(* CoDeSys 2.3.9.59 project: Indo_Tex.pro *)
(* Libraries: standard.lib 5.6.98 12:03:02, TcEtherCAT.lib 8.3.12 17:06:42, TcUtilities.lib 10.1.13 19:12:12, TcBase.lib 14.5.09 12:14:08, FB_Date_Time .lib 20.5.16 16:54:40, TcSystem.lib 27.2.12 14:08:36, TcBaseMath.lib 27.7.04 12:07:56, TcMath.lib 23.9.04 15:15:30, TcMC2.lib 13.9.17 10:18:38, SysLibVisu.lib 7.7.04 17:17:22, SysLibTargetVisu.lib 16.6.08 16:24:26, TcSystemCX.lib 7.9.16 12:51:26, COMlibV2.lib 1.8.08 13:22:48 *)

(* Global variable list: GVL_Alarm *)
VAR_GLOBAL
	RS_Error_1: RS_Error;
	RS_Error_2: RS_Error;
	RS_Error_3: RS_Error;
	RS_Error_4: RS_Error;
	RS_Error_5: RS_Error;
	RS_Error_6: RS_Error;
	RS_Error_7: RS_Error;

	bASealConvEnd1: BOOL;
	AlarmMess2: STRING(80);
	AlarmMess1: STRING(80);
	AlarWrap: STRING(80);
	CountMess: STRING(80);
	AlarmMessg: STRING(80);
	UnitASenSelet: UINT;
	SealingStep: INT;
	AlarmWrpConyMess: STRING(80);
	ConeMissAlarm: STRING(80);

	bAConeFeedCylRsError: BOOL;
	bAFwdCylRsError: BOOL;
	bAWrappingCylRsError: BOOL;
	bAWrappingCylRs1Error: BOOL;
	bAWrappingCylRs2Error: BOOL;
	bAWrappingCylRs3Error: BOOL;
	bAWrapCylRsErrorAuto: BOOL;
	bAError: BOOL;
	bASealTopCylRsError: BOOL;
	bASealBotCylRsError: BOOL;
	bASealTopBotCylRsError: BOOL;
	bASealSepXCylRsError: BOOL;
	bASealSepYCylRsError: BOOL;
	bASupplyPressureError: BOOL;
	HmiSupplyPressureMsg: STRING;
	bAFilmNotloaded: BOOL;
	bAConeMissAtSealConv: BOOL;
	bAEmergencyPressed: BOOL;
	bEmPopUp: BOOL;
	bAConeMissErrorAtWrpConv: BOOL;
	ConeAlignErr: BOOL;
	ConeMissAlarm1: STRING;
	ConeMissAlarm2: STRING;
	bAFlimNotLoaded: BOOL;
	bAPolythinSheetError: BOOL;
	bFilmErrClear: BOOL;
	bASepYAxisRsErrorChkBit: BOOL;
	bASepYAxisRsErrorChkBit1: BOOL;
	bABuzzer: BOOL;
	PressureChkTimer: TON;
	bAStop: BOOL;

	bAErrorChkBit: BOOL;
	bCheckWrappingSen: BOOL;
	bPloySheetSensError: BOOL;
	checkPolySheet2: BOOL;
	bAErrorChkBit2: BOOL;
	bCheckWrappingSen2: BOOL;
	bAErrorChkBit3: BOOL;
	bCheckWrappingSen3: BOOL;
	bWrapConvStopped2Temp: BOOL;
	SealingOk: BOOL;
	CycleComplete: BOOL;
	CycleComplete1: BOOL;
	SGrossWtNokMsg: STRING;

	SGrossWtCylEndSenErrMsg: STRING;
	bGrossWtCylEndSenError: BOOL;
END_VAR

(* Global variable list: GVL_Auto *)
VAR_GLOBAL
	bAutoModeOn: BOOL;
	bAPauseSeq: BOOL;
	bUnitBRowStopperStarted: BOOL;
	bUnitARowStopperStarted: BOOL;
	bAUnitAWeighOk: BOOL;
	bAConeFeedOver: BOOL;
	bAWrappingConvStart3: BOOL;
	bAWrappingConvStart1: BOOL;
	bAWrappingConvStart2: BOOL;
			bA3ConeWrappOver: BOOL;
	bA4thWrappOver: BOOL;
	bA6thConeWrappOver: BOOL;
	bA8thConeWrappOver: BOOL;
	bA6ConeWrappOver23: BOOL;
	AlarmMess: STRING(80);
	bAWrappingCone123OnAuto: BOOL;
	bAFwdPistonComp1: BOOL;
	bAFwdPistonComp2: BOOL;
	bAFwdPistonComp3: BOOL;
	bAConvFirstStart: BOOL;
	UnitACompleteCheckCount: CTU;
	bRetUnitAStart: BOOL;
	bRetUnitBStart: BOOL;
	bAUnitBWeighOk: BOOL;
	(*UnitAConeCompChkCount: CTU;*)
	iSensorOnVal: USINT;
	bFwdPistonStartTemp: BOOL;
	bConeMiss1AtWrapConv: BOOL;
	bConeMiss2tWrapConv: BOOL;
	bConeMiss2AtWrapConv: BOOL;
	ConeMissbit: BOOL;
	CTU_1: CTU;
	bAPauseEnable: BOOL;
	SealComDlyTemp: TIME;
	bAMcStartInAuto: BOOL;
	bPauseExtend: BOOL;
	bAutoModeOff: BOOL;
	iTotalNoOfCones: BOOL;
	iATotalNoOfCones: INT;
	bAMcReady: BOOL;
	bAMcRunninig: BOOL;
	bAFilmLoaded: BOOL;
	bAWrapConStart: BOOL;
	bA3ConeWrappOverTemp: BOOL;
	bABypassOn: BOOL;
	bIntialAckBit: BOOL;
	ConeInComplete: BOOL;
	ConeInCompletetest: BOOL;
	ConeInCompleteTestbitB: BOOL;
	bUnitACounterDIsable: BOOL;
	ConeInCompleteA: BOOL;
	bAOneMinConvStart: BOOL;
	bAWrapwait: BOOL;
END_VAR

(* Global variable list: GVL_Hmi *)
VAR_GLOBAL
	bStopHmi: BOOL;
	bInitializeHmi: BOOL;

	HMIFeedPiston: STRING(80);
	HMIWrapPiston1: STRING(80);
	HMIWrapPiston2: STRING(80);
	HMIWrapPiston3: STRING(80);
	HMIForwdPiston:STRING(80);
	HMISealBotPiston:STRING(80);
	HMISealTopPiston:STRING(80);
	HmiXAxisPiston:STRING(80);
	HmiYAxisPiston:STRING(80);
	bErrorReset: BOOL;
	bPauseHmi: BOOL;
	bResumeHmi: BOOL;
	bResetTemp: BOOL;
	bHmiAck: BOOL;

	b18ConeModelHmi: BOOL;
	b12ConeModelHmi:BOOL;
	b24ConeModelHmi: BOOL;
	b32ConeModelHmi: BOOL;
	sAMcModeStatus: STRING;
	bAUnitBConeCrossed: BOOL;
	bAInializeStarted: BOOL;
	PopUp: BOOL;
	sAlarmStatus: STRING;
	bNegTolDisableHMI: BOOL;
	bNegTolEnableHMI: BOOL;
	bPrssurePopUp: BOOL;
	UnitAConeCountHMI: INT;
	UnitBConeCountHMI: INT;
	b16ConeModelHmi: BOOL;
	WrapConeSenDetMes: STRING;
	bAmberbit2: BOOL;
	Pgm_NoHmi: INT;
	FileCreateTemp: BOOL;
	bACyclePass: BOOL;
	iCartoNoHmi: STRING;
	(*iLotNoHmi: STRING;*)
	var_1: REAL;
	var_5: REAL;
	LogYear: STRING;
	LogMonth: STRING;
	logDay: STRING;
	sTIME: STRING;
	sDATEFinal: STRING;
	DateTimeVar: STRING;
	wTodayToHmi: STRING;
	bInterlockInitial_2: BOOL;
	sMessage: STRING;
	bReadGWieght: BOOL;
	bAReset_all_error: BOOL;








	LotASelected: BOOL;
	LotACartonNo: INT;
	LotBSelected: BOOL;
	LotBCartonNo: INT;
	LotCSelected: BOOL;
	LotDSelected: BOOL;
	LotESelected: BOOL;
	LotFSelected: BOOL;
	LotCCartonNo: INT;
	LotDCartonNo:  INT;
	LotECartonNo:  INT;
	LotFCartonNo: INT;
	LotA: INT;

	LotB: INT;

	LotC: INT;

	LotAHmi: BOOL;
	LotBHmi: BOOL;
	LotCHmi: BOOL;
	CurrentCartonNo:INT;
	LotNoChange: BOOL;
	ParametesSave: BOOL;
END_VAR

VAR_GLOBAL RETAIN
(*VAR_GLOBAL PERSISTENT*)
	b12ConeModelSelected AT %Q*: BOOL;
	b18ConeModelSelected AT %Q*: BOOL;
	b24ConeModelSelected AT %Q*: BOOL;
	b32ConeModelSelected AT %Q*: BOOL;
	rSealCompDlyHmi AT %Q*: REAL;
	iNetTolHmi AT %Q*: REAL;
	iNetWtHmi AT %Q*: REAL;
	iLotNoHmi AT %Q*: STRING;
	iWorkOrderNoHmi AT %Q*:STRING;
	NegToleranceEnabled AT %Q*: BOOL;
	b16ConeModelSelected AT %Q*: BOOL;
	ProgramNoHmi AT %Q*: INT;
	CountCodeHmi AT %Q*: STRING(80);
	CartonNoHmi AT %Q*: INT;
	DefaultNetWeightHmi AT %Q*: REAL;
	DefaultGrossWeightHmi AT %Q*: REAL;
	EmptyConeWt AT %Q*: REAL;
	BlendHmi AT %Q*: STRING(80);
	ShadeHmi AT %Q*: STRING(80);
	ConeTipHmi AT %Q*: STRING(80);
	ConeNettHmi AT %Q*: STRING(80);
	ConeLengthHmi AT %Q*: REAL;
	Cones:INT;
	Dom_ExpHmi AT %Q*: STRING(80);
	PackTypeHmi AT %Q*: STRING(80);
	ItemCodeHmi AT %Q*: STRING(80);
	IssueDesp AT %Q*: STRING(80);
	Location AT %Q*: STRING(80);
	Description AT %Q*: STRING(80);
	Remarks AT %Q*: STRING(80);
	Fyear AT %Q*: STRING(80);
	AvgCount AT %Q*: STRING(80);
	TareWeight AT %Q*: REAL;
	BarCode AT %Q*: STRING(80);
	WorkFlag AT %Q*: STRING(80);
END_VAR

(* Global variable list: GVL_Inputs *)
VAR_GLOBAL


(******************EL1809-1(Main)*********************)

	bIConeFeedingPistonHome AT %IX0.0: BOOL;
	bIConeFeedingPistonEnd AT %IX0.1: BOOL;
	bIConeOrientationTop AT %IX0.2: BOOL;
	bIForwardPistonHome AT %IX0.3: BOOL;
	bIForwardPistonEnd AT %IX0.4: BOOL;
	bIWrappingConeDeductionSen AT %IX0.5: BOOL;
	bISpare1 AT %IX0.6: BOOL;
	bISpare2 AT %IX0.7: BOOL;
	bISpare3 AT %IX1.0: BOOL;
	bIWrappingChannelPiston1_Home AT %IX1.1: BOOL;
	bIWrappingChannelPiston1_End AT %IX1.2: BOOL;
	bIWrappingChannelPiston2_Home AT %IX1.3: BOOL;
	bIWrappingChannelPiston2_End AT %IX1.4: BOOL;
	bIWrappingChannelPiston3_Home AT %IX1.5: BOOL;
	bIWrappingChannelPiston3_End AT %IX1.6: BOOL;
	bIWrappingCone1 AT %IX1.7:BOOL;

(******************EL1809-2(Main)*********************)

	bIWrappingCone2 AT %IX2.0: BOOL;
	bIWrappingCone3 AT %IX2.1: BOOL;
	bIWrappingFilmTensionPlate_1 AT %IX2.2: BOOL;
	bIWrappingFilmTensionPlate_2 AT %IX2.3: BOOL;
	bIWrappingFilmTensionPlate_3 AT %IX2.4: BOOL;
	bISealingTopPistonHome AT %IX2.5: BOOL;
	bISealingTopPistonEnd AT %IX2.6: BOOL;
	bISealingBottomPistonHome AT %IX2.7: BOOL;
	bISealingBottomPistonEnd AT %IX3.0: BOOL;
	bIConeCountSensor AT %IX3.1: BOOL;
	bISealingSeparatorYAxisHome AT %IX3.2: BOOL;
	bISealingSeparatorYAxisEnd AT %IX3.3: BOOL;
	bISealingSeparatorXAxisHome AT %IX3.4: BOOL;
	bISealingSeparatorXAxisEnd AT %IX3.5: BOOL;
	bIManualSealing AT %IX3.6: BOOL;
	bIPressureSwitch  AT %IX3.7: BOOL;

(******************EL1809-3(Main)*********************)

	bISpare4  AT %IX4.0: BOOL;
	bISpare5   AT %IX4.1: BOOL;
	bIUnitA_RowStopperHome   AT %IX4.2: BOOL;
	bIUnitA_RowStopperEnd AT %IX4.3: BOOL;
	bIUnitB_RowStopperHome AT %IX4.4: BOOL;
	bIUnitB_RowStopperEnd AT %IX4.5: BOOL;
	bIUnitA_StartPB AT %IX4.6: BOOL;
	bIUnitB_StartPB AT %IX4.7:BOOL;
	bIUnitAConeDetection4 AT %IX5.0:BOOL;
	bIUnitBConeDetection4 AT %IX5.1:BOOL;
	bIUnitAConeDetection1 AT %IX5.2:BOOL;
	bIUnitAConeDetection2 AT %IX5.3:BOOL;
	bIUnitAConeDetection3 AT %IX5.4:BOOL;
	bIUnitAConeCrossing AT %IX5.5:BOOL;
	bIUnitBConeDetection1 AT %IX5.6:BOOL;
	bIUnitBConeDetection2 AT %IX5.7:BOOL;

(******************EL1809-4(Main)*********************)

	bIUnitBConeDetection3 AT %IX6.0:BOOL;
	bIUnitBConeCrossing AT %IX6.1:BOOL;
	bIAutoManual AT %IX6.2:BOOL;
	bIMCStart AT %IX6.3:BOOL;
	bIMCStop AT %IX6.4:BOOL;
	bIKeySwitch AT %IX6.5:BOOL;
	bIEmergency AT %IX6.6:BOOL;
	bIUnitA_RowStopperMiddle AT %IX6.7:BOOL;

	bIUnitB_RowStopperMiddle AT %IX7.0: BOOL;
	bIGross_Crossing_Input  AT %IX7.1: BOOL;
	bIGross_Weight_Stop AT %IX7.2: BOOL;
	bIGross_Cyl_Home AT %IX7.3: BOOL;
	bIGross_Cyl_End AT %IX7.4: BOOL;
	bISpare12 AT %IX7.5: BOOL;
	bISpare13 AT %IX7.6: BOOL;
	bISpare14 AT %IX7.7: BOOL;
END_VAR

(* Global variable list: GVL_Manual *)
VAR_GLOBAL




		bQMConeFeedingPistonValve :BOOL;
		bQMForwardPistonValve  :BOOL;
		bQMReversePistonValve :BOOL;
		bQMWrappingChannelPistonValve1:BOOL;
		bQMWrappingChannelPistonValve2:BOOL;
		bQMWrappingChannelPistonValve3 :BOOL;
		bQMSealingTopPistonValve :BOOL;
		bQMSealingBottomPistonValve:BOOL;


		bQMFeedingConveyorMotor :BOOL;
		bQMWrappingConveyorMotor :BOOL;
		bQMSealingConveyorMotor :BOOL;
		bQMMatrixConveyorMotor :BOOL;
		bQMFilmRollerMotor1 :BOOL;
		bQMFilmRollerMotor2 :BOOL;
		bQMFilmRollerMotor3 :BOOL;




		bQMRowStopperMotorForward  :BOOL;
		bQMRowStopperMotorReverse:BOOL;
		bQMColumnStopperMotorForward :BOOL;
		bQMColumnStopperMotorReverse:BOOL;
		bQMSealingSeparatorYAxisPistonValve :BOOL;
		bQMSealingSeparatorXAxisPistonValve :BOOL;
		bQMConeTiltingPistonValve :BOOL;
		bQMColumnPushPistonValve:BOOL;

		bQMSeparatorHorizontalPistonValveFwd :BOOL;
		bQMSeparatorVerticalPistonValve :BOOL;
		bQMCartonFeedingPistonValve :BOOL;
		bQMConeEjectionPistonValve :BOOL;
		bQMLengthTightPistonValve :BOOL;
		bQMBreadthTightPistonValve:BOOL;
		bQMEmptyCartonConveyorMotor :BOOL;
		bQMCartonConveyorMotor :BOOL;





		bQMVacuumPistonValve  :BOOL;
		bQMSeparatorHorizontalPistonValveRev  :BOOL;
		bQMSpare1  :BOOL;
		bQMSpare2 :BOOL;


	bQMUnitA_LiftPistonValve:BOOL;
	bQMUnitB_LiftPistonValve: BOOL;
	bQMUnitA_RowStopperMotorForward :BOOL;
	bQMUnitA_RowStopperMotorReverse :BOOL;
	bQMUnitB_RowStopperMotorForward :BOOL;
	bQMUnitB_RowStopperMotorReverse:BOOL;
	bQMUnitC_FullCartonConveyor :BOOL;
	bQMUnitC_LiftPistonValve :BOOL;


	bUA_LiftCylOnHmi: BOOL;
	bUA_LiftCylOffHmi: BOOL;
	bUB_LiftCylOnHmi: BOOL;
	bUB_LiftCylOffHmi: BOOL;
	bUA_RowStopperMotorFwd: BOOL;
	bUA_RowStopperMotorFwdOnHmi: BOOL;
	bUA_RowStopperMotorFwdOffHmi: BOOL;
	bUA_RowStopperMotorRevOnHmi: BOOL;
	bUB_RowStopperMotorFwdOnHmi: BOOL;
	bUB_RowStopperMotorRevOnHmi: BOOL;
	bUC_FullCartonConv: BOOL;
	bUC_FullCartonConvOnHmi: BOOL;
	bUC_FullCartonConvOffHmi: BOOL;
	bUC_LiftCylOnHmi: BOOL;
	bUC_LiftCylOffHmi: BOOL;

	bCFPistonOnHmi: BOOL;
	bCFPistonOffHmi: BOOL;
	bFPValveOnHmi:BOOL;
	bFPValveOffHmi:BOOL;
	bRPValveOnHmi:BOOL;
	bRPValveOffHmi:BOOL;
	bWrappingCPV1OnHmi:BOOL;
	bWrappingCPV1OffHmi:BOOL;
	bWrappingCPV2OnHmi:BOOL;
	bWrappingCPV2OffHmi:BOOL;
	bWrappingCPV3OnHmi:BOOL;
	bWrappingCPV3OffHmi:BOOL;
	bSealingTopPVOnHmi:BOOL;
	bSealingTopPVOffHmi:BOOL;
	bSealingBottomPVOnHmi:BOOL;
	bSealingBottomPVOffHmi:BOOL;
	bFCMotorOnHmi:BOOL;
	bFCMotorOffHmi:BOOL;
	bWCMotorOnHmi:BOOL;
	bWCMotorOffHmi:BOOL;

	bSCMotorOnHmi: BOOL;
	bSCMotorOffHmi: BOOL;
	bMCMotorOnHmi: BOOL;
	bMCMotorOffHmi: BOOL;
	bFRMotor2OnHmi: BOOL;
	bFRMotor2OffHmi: BOOL;
	bFRMotor1OnHmi: BOOL;
	bFRMotor1OffHmi: BOOL;
	bFRMotor3OnHmi: BOOL;
	bFRMotor3OffHmi: BOOL;
	bRSMotorForwardOnHmi: BOOL;
	bRSMotorForwardOffHmi: BOOL;
	bRSMotorRevOnHmi: BOOL;
	bRSMotorRevOffHmi: BOOL;
	bCSMotorFwdOnHmi: BOOL;
	bCSMotorFwdOffHmi: BOOL;
	bCSMotorRevOnHmi: BOOL;
	bCSMotorRevOffHmi: BOOL;
	bSSYAxisPistonValveOnHmi: BOOL;
	bSSYAxisPistonValveOffHmi: BOOL;
	bSSXAxisPistonValveOnHmi: BOOL;
	bSSXAxisPistonValveOffHmi: BOOL;
	bCTPistonValveOnHmi: BOOL;
	bCTPistonValveOffHmi: BOOL;
	bCPushPistonValveOnHmi: BOOL;
	bCPushPistonValveOffHmi: BOOL;
	bSHPistonValveOnHmi: BOOL;
	bSHPistonValveOffHmi: BOOL;
	bSVPistonValveOnHmi: BOOL;
	bSVPistonValveOffHmi: BOOL;
	bCPistonValveOnHmi: BOOL;
	bCPistonValveOffHmi: BOOL;
	bCEPistonValveOnHmi: BOOL;
	bCEPistonValveOffHmi: BOOL;
	bLTPistonValveOnHmi: BOOL;
	bLTPistonValveOffHmi: BOOL;
	bBTightPistonValveOnHmi: BOOL;
	bBTightPistonValveOffHmi: BOOL;
	bECCMotorOnHmi: BOOL;
	bECCMotorOffHmi: BOOL;
	bCCMotorOnHmi: BOOL;
	bCCMotorOffHmi: BOOL;
	bVPValveOnHmi: BOOL;
	bVPValveOffHmi: BOOL;
	bSHPistonValveREVOnHmi: BOOL;
	bSHPistonValveREVOffHmi: BOOL;
	bQMSeparatorHorizontalPistonValveFOR: BOOL;
	bQMColumnPushPistonValveY: BOOL;
	bCPushPistonValveYOnHmi: BOOL;
	bCPushPistonValveYOffHmi: BOOL;
	bMManualSealOn: BOOL;
	bQMLengthPistonValve: BOOL;
	bQMBreathPistonValve: BOOL;
	bQMGrossWtPiston: BOOL;
	bQMRollerConvMotor: BOOL;
	bGWPistonOffHmi1: BOOL;
	bManualModeOn: BOOL;
END_VAR

(* Global variable list: GVL_OutputFlags *)
VAR_GLOBAL



		bQAConeFeedingPistonValve  :BOOL;
		bQAForwardPistonValve  :BOOL;
		bQAWrappingChannelPistonValve1  :BOOL;
		bQAWrappingChannelPistonValve2 :BOOL;
		bQAWrappingChannelPistonValve3:BOOL;
		bQASealingTopPistonValve :BOOL;
		bQASealingBottomPistonValve:BOOL;
		bQASealingSeparatorYAxisPistonValve :BOOL;

		bQASealingSeparatorXAxisPistonValve :BOOL;
		bQAFeedingConveyorMotor :BOOL;
		bQAWrappingConveyorMotor:BOOL;
		bQAFilmRollerMotor1 :BOOL;
		bQAFilmRollerMotor2 :BOOL;
		bQAFilmRollerMotor3 :BOOL;
		bQASealingConveyorMotorFWD :BOOL;







		bQAUnitARowStopperMotorFwd  :BOOL;
		bQAUnitARowStopperMotorRev  :BOOL;
		bQAUnitBRowStopperMotorFwd  :BOOL;
		bQAUnitBRowStopperMotorRev :BOOL;
		bQAUnitAWeightOkLamp :BOOL;
		bQAUnitAWeightNokLamp  :BOOL;
		bQAUnitBWeightOkLamp :BOOL;
		bQAUnitBWeightNokLamp  :BOOL;


		bQABuzzer :BOOL;
		bQASpare1 :BOOL;
		bQASpare2 :BOOL;
		bQASpare3  :BOOL;
		bQASpare4  :BOOL;

	bQAUnitA_RowStopperMotorReverse1: BOOL;
	bQAUnitA_RowStopperMotorForward1: BOOL;
	bQASealingConveyorMotor: BOOL;

	bQASealingConveyor1: BOOL;
	bQAWrappingConveyorMotor1: BOOL;
	bQAWrappingConveyorMotor2: BOOL;
	bQAWrappingConveyorMotor3: BOOL;
	bQAAmber: BOOL;
	bQAGreen: BOOL;
	bQARed: BOOL;
	(*UnitBCompleteCheckCount: CTU;*)
END_VAR

(* Global variable list: GVL_Outputs *)
VAR_GLOBAL

		(*===============EL2809-1(Main) ===========*)


		bQConeFeedingPistonValve AT %QX0.0 :BOOL;
		bQForwardPistonValve AT %QX0.1 :BOOL;
		bQWrappingChannelPistonValve1 AT %QX0.2 :BOOL;
		bQWrappingChannelPistonValve2 AT %QX0.3:BOOL;
		bQWrappingChannelPistonValve3 AT %QX0.4:BOOL;
		bQSealingTopPistonValve AT %QX0.5:BOOL;
		bQSealingBottomPistonValve AT %QX0.6:BOOL;
		bQSealingSeparatorYAxisPistonValve AT %QX0.7:BOOL;

		bQSealingSeparatorXAxisPistonValve  AT %QX1.0:BOOL;
		bQFeedingConveyorMotor AT %QX1.1:BOOL;
		bQWrappingConveyorMotor AT %QX1.2:BOOL;
		bQFilmRollerMotor1 AT %QX1.3:BOOL;
		bQFilmRollerMotor2 AT %QX1.4:BOOL;
		bQFilmRollerMotor3 AT %QX1.5:BOOL;
		bQSealingConveyorMotorFWD AT %QX1.6:BOOL;
		bQUnitARowStopperMotorFwd AT %QX1.7:BOOL;



		(*===============EL2809-2( Main )===========*)



		bQUnitARowStopperMotorRev AT %QX2.0 :BOOL;
		bQUnitBRowStopperMotorFwd AT %QX2.1 :BOOL;
		bQUnitBRowStopperMotorRev AT %QX2.2:BOOL;
		bQUnitAWeightOkLamp  AT %QX2.3:BOOL;
		bQUnitAWeightNokLamp  AT %QX2.4:BOOL;
		bQUnitBWeightOkLamp  AT %QX2.5:BOOL;
		bQUnitBWeightNokLamp  AT %QX2.6:BOOL;
		bQTLGreen AT %QX2.7 :BOOL;

		bQTLAmber AT %QX3.0 :BOOL;
		bQTLRed AT %QX3.1 :BOOL;
		bQBuzzer AT %QX3.2 :BOOL;
		bQGross_Roller_On AT %QX3.3:BOOL;
		bQGross_Cylinder_On AT %QX3.4:BOOL;
		bQSpare3 AT %QX3.5:BOOL;
		bQSpare4  AT %QX3.6:BOOL;
		bQSpare5  AT %QX3.7:BOOL;



		(*===============EL2008-2( Main )===========*)








END_VAR

(* Global variable list: GVL_Reset *)
VAR_GLOBAL
	bQRForwardPistonValve: BOOL;
	bQRWrappingChannelPistonValve2: BOOL;
	bQRWrappingChannelPistonValve3: BOOL;
	bQRSealingTopPistonValve: BOOL;
	bQRSealingSeparatorYAxisPistonValve: BOOL;
	bQRSealingSeparatorXAxisPistonValve: BOOL;
	bQRSealingConveyorMotor: BOOL;
	bQRWrappingChannelPistonValve1: BOOL;
	bQRWrappingConveyorMotor: BOOL;
	bFwdPistonRst: BOOL;
	bARWrappingCone123OnRst: BOOL;

	bAR3ConeWrappOver: BOOL;
	bSaelUnitIntOver: BOOL;
	bWCSStart1: BOOL;
	bAInitializeSeq: BOOL;
	bSealConvIntOver: BOOL;
	sSealConvStatus: STRING;
	sWrapConvStatus: STRING;
	bWrpConvIntOver: BOOL;
END_VAR

(* Global variable list: GVL_Serial *)
VAR_GLOBAL
	rRetUnitBWeight: REAL;
	rRetUnitAWeight: REAL;
	COMin_COMPort AT %I*: EL6inData22B;
	COMOut_COMPort AT %Q*: EL6outData22B;
	TxBuffer1: ComBuffer;
	RxBuffer1: ComBuffer;

	COMin_2_COMport_2 AT %I*: EL6inData22B;
	COMout_2_COMport_2 AT %Q*: EL6outData22B;
	TxBuffer2: ComBuffer;
	RxBuffer2: ComBuffer;

	COMin_3_COMport_3 AT %I*: EL6inData22B;
	COMout_3_COMport_3 AT %Q*: EL6outData22B;
	TxBuffer3: ComBuffer;
	RxBuffer3: ComBuffer;

	COMin_4_COMport_4 AT %I*: EL6inData22B;
	COMout_4_COMport_4 AT %Q*: EL6outData22B;
	TxBuffer4: ComBuffer;
	RxBuffer4: ComBuffer;

	rGrossWeight: REAL;
	bGrossWieghtNokTemp: BOOL;
	bGrossWieghtOk: BOOL;
	bQAGrossWieghtOkIndi: BOOL;
	bGrossWieghtNOk: BOOL;
	GrossWtReedSwBit: BOOL;
	bIGrossWtPistonHome: BOOL;
	bAGrossWtHomeSenRsError: BOOL;
	One_Min_Conv_1: INT;
	rGrossWeighToReport: REAL;
END_VAR

VAR_GLOBAL PERSISTENT
	sGrosswt AT %Q*: REAL;
	sGrossTol AT %Q*: REAL;
END_VAR

(* Global variable list: PARAMETERS *)
VAR_GLOBAL
	SAVE: BOOL;
	TotalCones: DINT;
	iBagCount: DINT;
	LOAD: BOOL;
	sBagNoRep: STRING;
	sDayMonthYearDate: STRING;
	PROCESSCOMPLETE: BOOL;



	PRGNO_LOAD: DINT;
	NegTolEnableHmi AT %Q*: BOOL;
	NegTol1EnableHmi AT %Q*: BOOL;
	NegTol2EnableHmi AT %Q*: BOOL;
	NegTol3EnableHmi AT %Q*: BOOL;
	NegTol4EnableHmi AT %Q*: BOOL;
	NegTol5EnableHmi AT %Q*: BOOL;

	PRGNO_DIS AT %Q*: DINT;
	COUNT_DIS AT %Q*: STRING(80);
	DETAILS_DIS AT %Q*: STRING(80);
	LOTNO_DIS AT %Q*: STRING(80);
	CARTONNO_DIS AT %Q*: DINT;
	WORKORDERNO_DIS:STRING;
	BLEND_DIS:STRING;
	SHADE_DIS:STRING;
	CONETIP_DIS:STRING;
	CONELENGTH_DIS:REAL;
	CONENETWT_DIS:REAL;
	DFLTNETWT_DIS AT %Q*: REAL;
	NETWTTOL_DIS AT %Q*: REAL;
	DFLTGROSSWT_DIS AT %Q*: REAL;
	GROSSWTTOL_DIS AT %Q*: REAL;
	NegTol_DIS AT %Q*: REAL;



	PRGNO AT %Q*: DINT;
	COUNT AT %Q*: STRING(80);
	DETAILS AT %Q*: STRING(80);
	LOTNO AT %Q*: STRING(80);
	CARTONNO AT %Q*: DINT;
	WORKORDERNO:STRING;
	BLEND:STRING;
	SHADE:STRING;
	CONETIP:STRING;
	CONELENGTH:REAL;
	CONENETWT:REAL;
	DFLTNETWT AT %Q*: REAL;
	NETWTTOL AT %Q*: REAL;
	DFLTGROSSWT AT %Q*: REAL;
	GROSSWTTOL AT %Q*: REAL;
	NegTol AT %Q*: REAL;

	PRGNO1 AT %Q*: DINT;
	COUNT1 AT %Q*: STRING(80);
	DETAILS1 AT %Q*: STRING(80);
	LOTNO1 AT %Q*: STRING(80);
	CARTONNO1 AT %Q*: DINT;
	WORKORDERNO1:STRING;
	BLEND1:STRING;
	SHADE1:STRING;
	CONETIP1:STRING;
	CONELENGTH1:REAL;
	CONENETWT1:REAL;
	DFLTNETWT1 AT %Q*: REAL;
	NETWTTOL1 AT %Q*: REAL;
	DFLTGROSSWT1 AT %Q*: REAL;
	GROSSWTTOL1 AT %Q*: REAL;
	NegTol1 AT %Q*: REAL;

	PRGNO2 AT %Q*: DINT;
	COUNT2 AT %Q*: STRING(80);
	DETAILS2 AT %Q*: STRING(80);
	LOTNO2 AT %Q*: STRING(80);
	CARTONNO2 AT %Q*: DINT;
	WORKORDERNO2:STRING;
	BLEND2:STRING;
	SHADE2:STRING;
	CONETIP2:STRING;
	CONELENGTH2:REAL;
	CONENETWT2:REAL;
	DFLTNETWT2 AT %Q*: REAL;
	NETWTTOL2 AT %Q*: REAL;
	DFLTGROSSWT2 AT %Q*: REAL;
	GROSSWTTOL2 AT %Q*: REAL;
	NegTol2 AT %Q*: REAL;

	PRGNO3 AT %Q*: DINT;
	COUNT3 AT %Q*: STRING(80);
	DETAILS3 AT %Q*: STRING(80);
	LOTNO3 AT %Q*: STRING(80);
	CARTONNO3 AT %Q*: DINT;
	WORKORDERNO3:STRING;
	BLEND3:STRING;
	SHADE3:STRING;
	CONETIP3:STRING;
	CONELENGTH3:REAL;
	CONENETWT3:REAL;
	DFLTNETWT3 AT %Q*: REAL;
	NETWTTOL3 AT %Q*: REAL;
	DFLTGROSSWT3 AT %Q*: REAL;
	GROSSWTTOL3 AT %Q*: REAL;
	NegTol3 AT %Q*: REAL;

	PRGNO4 AT %Q*: DINT;
	COUNT4 AT %Q*: STRING(80);
	DETAILS4 AT %Q*: STRING(80);
	LOTNO4 AT %Q*: STRING(80);
	CARTONNO4 AT %Q*: DINT;
	WORKORDERNO4:STRING;
	BLEND4:STRING;
	SHADE4:STRING;
	CONETIP4:STRING;
	CONELENGTH4:REAL;
	CONENETWT4:REAL;
	DFLTNETWT4 AT %Q*: REAL;
	NETWTTOL4 AT %Q*: REAL;
	DFLTGROSSWT4 AT %Q*: REAL;
	GROSSWTTOL4 AT %Q*: REAL;
	NegTol4 AT %Q*: REAL;


	PRGNO5 AT %Q*: DINT;
	COUNT5 AT %Q*: STRING(80);
	DETAILS5 AT %Q*: STRING(80);
	LOTNO5 AT %Q*: STRING(80);
	CARTONNO5 AT %Q*: DINT;
	WORKORDERNO5:STRING;
	BLEND5:STRING;
	SHADE5:STRING;
	CONETIP5:STRING;
	CONELENGTH5:REAL;
	CONENETWT5:REAL;
	DFLTNETWT5 AT %Q*: REAL;
	NETWTTOL5 AT %Q*: REAL;
	DFLTGROSSWT5 AT %Q*: REAL;
	GROSSWTTOL5 AT %Q*: REAL;
	NegTol5 AT %Q*: REAL;


	PRGNO6:DINT;
	COUNT6:STRING;
	DETAILS6:STRING;
	LOTNO6:STRING;
	CARTONNO6:DINT;
	WORKORDERNO6:STRING;
	BLEND6:STRING;
	SHADE6:STRING;
	CONETIP6:STRING;
	CONELENGTH6:REAL;
	CONENETWT6:REAL;
	DFLTNETWT6:REAL;
	NETWTTOL6:REAL;
	DFLTGROSSWT6:REAL;
	GROSSWTTOL6:REAL;


	PRGNO7:DINT;
	COUNT7:STRING;
	DETAILS7:STRING;
	LOTNO7:STRING;
	CARTONNO7:DINT;
	WORKORDERNO7:STRING;
	BLEND7:STRING;
	SHADE7:STRING;
	CONETIP7:STRING;
	CONELENGTH7:REAL;
	CONENETWT7:REAL;
	DFLTNETWT7:REAL;
	NETWTTOL7:REAL;
	DFLTGROSSWT7:REAL;
	GROSSWTTOL7:REAL;


	PRGNO8:DINT;
	COUNT8:STRING;
	DETAILS8:STRING;
	LOTNO8:STRING;
	CARTONNO8:DINT;
	WORKORDERNO8:STRING;
	BLEND8:STRING;
	SHADE8:STRING;
	CONETIP8:STRING;
	CONELENGTH8:REAL;
	CONENETWT8:REAL;
	DFLTNETWT8:REAL;
	NETWTTOL8:REAL;
	DFLTGROSSWT8:REAL;
	GROSSWTTOL8:REAL;


	PRGNO9:DINT;
	COUNT9:STRING;
	DETAILS9:STRING;
	LOTNO9:STRING;
	CARTONNO9:DINT;
	WORKORDERNO9:STRING;
	BLEND9:STRING;
	SHADE9:STRING;
	CONETIP9:STRING;
	CONELENGTH9:REAL;
	CONENETWT9:REAL;
	DFLTNETWT9:REAL;
	NETWTTOL9:REAL;
	DFLTGROSSWT9:REAL;
	GROSSWTTOL9:REAL;


	PRGNO10:DINT;
	COUNT10:STRING;
	DETAILS10:STRING;
	LOTNO10:STRING;
	CARTONNO10:DINT;
	WORKORDERNO10:STRING;
	BLEND10:STRING;
	SHADE10:STRING;
	CONETIP10:STRING;
	CONELENGTH10:REAL;
	CONENETWT10:REAL;
	DFLTNETWT10:REAL;
	NETWTTOL10:REAL;
	DFLTGROSSWT10:REAL;
	GROSSWTTOL10:REAL;

	PRG1RUNNING AT %Q*: BOOL;
	PRG2RUNNING AT %Q*: BOOL;
	PRG3RUNNING AT %Q*: BOOL;
	PRG4RUNNING AT %Q*: BOOL;
	PRG5RUNNING AT %Q*: BOOL;
	PRG6RUNNING: BOOL;
	PRG7RUNNING: BOOL;
	PRG8RUNNING: BOOL;
	PRG9RUNNING: BOOL;
	PRG10RUNNING: BOOL;
	PRINTENABLE: BOOL;
	PRINTENABLED: BOOL;

	DfltWtPrint: BOOL;
	DfltGrossWtPrint_En: BOOL;
	GrossWtPrintDflt: BOOL;
	NetwtPrint: STRING;
	GrosswtPrint: STRING;

	ReportPath: STRING;
	sDayF1: STRING;
	sMonthF1: STRING;
	sDayMonth1: STRING;

	ReportPath_Final_2: STRING;
	FB_DateTime_2: FB_DateTime;
	sDaateReport: STRING;







	sDayMonthYear1: STRING;

	sDayMonthYear: STRING;
	ReportPath_Final_1: STRING;
	ReportPath_Final: STRING;
END_VAR

(* Global variable list: PRINT *)
VAR_GLOBAL

	ProductionData_Print: STRING(255);
	ProductionDataValues_Print: STRING(255);
	ProductionDataValues_Print_Com:STRING(255);
	PrintOk: BOOL;
	PrintEnableHmi: BOOL;
	PrintValue: INT;
	bANewDay: BOOL;
	ProductionDataValues_IndoPrint: STRING(255);
	ProductionData_IndoPrint: STRING(255);
	ProductionDataError_IndoPrint: STRING(255);

	ProductionData_IndoPrint2:STRING(255);
	ProductionDataError_IndoPrint2:STRING(255);
	ProductionDataValues_IndoPrint_Com:STRING(255);
		ProductionDataValuesError_IndoPrint_Com:STRING(255);
	ProductionData_IndoPrint11 : ProductionData_IndoPrint1;

	SerialNoError: DINT;




	ReportPathError: STRING;
	ReportPath_FinalError: STRING;
	ReportPath_Final_1Error: STRING;
	ReportPath_Final_2Error: STRING;
	stStation1_ProductionData:Production_Data;
	sHourPreFix: STRING;
	sHou: STRING;
	sDayPreFix: STRING;
	sDay: STRING;
	sMonthPreFix: STRING;
	sMonth: STRING;
	sDayF: STRING;
	sMonthF: STRING;
	sDayMonth: STRING;

	SerialNo AT %Q*: DINT;
	BagSerialNo: DINT;
	ReportSave: BOOL;
	wTodayToHmiFinal: STRING;
	Default_NetWeight_Report: STRING;
	Default_GrossWeight_Report: STRING;
	Actual_NetWeight_Report: STRING;
	Actual_GrossWeight_Report: STRING;
	negativetolerance AT %Q*: BOOL;
	DefaultNetWt AT %Q*: REAL;
	NetWtTolRep AT %Q*: REAL;
	DefaultGrossWt AT %Q*: REAL;
	GrossWtTolRep AT %Q*: REAL;


END_VAR

(* Global variable list: TwinCAT_Configuration *)
(* Generated automatically by TwinCAT - (read only) *)
VAR_CONFIG
	.b12ConeModelSelected AT %QX288.0 : BOOL;	(*  ~ {LinkedWith:TIID^Device 3 (NOV/DP-RAM)^Outputs^Model_1} *)
	.b18ConeModelSelected AT %QX288.1 : BOOL;	(*  ~ {LinkedWith:TIID^Device 3 (NOV/DP-RAM)^Outputs^Model_2} *)
	.b24ConeModelSelected AT %QX288.2 : BOOL;	(*  ~ {LinkedWith:TIID^Device 3 (NOV/DP-RAM)^Outputs^Model_3} *)
	.b32ConeModelSelected AT %QX288.3 : BOOL;	(*  ~ {LinkedWith:TIID^Device 3 (NOV/DP-RAM)^Outputs^Model_4} *)
	.rSealCompDlyHmi AT %QB52 : REAL;	(*  ~ {LinkedWith:TIID^Device 3 (NOV/DP-RAM)^Outputs^SealDly} *)
	.iNetTolHmi AT %QB56 : REAL;	(*  ~ {LinkedWith:TIID^Device 3 (NOV/DP-RAM)^Outputs^NetWtTol} *)
	.iNetWtHmi AT %QB60 : REAL;	(*  ~ {LinkedWith:TIID^Device 3 (NOV/DP-RAM)^Outputs^NetWt} *)
	.iLotNoHmi AT %QB64 : STRING(80);	(*  ~ {LinkedWith:TIID^Device 3 (NOV/DP-RAM)^Outputs^Var 339} *)
	.iWorkOrderNoHmi AT %QB148 : STRING(80);	(*  ~ {LinkedWith:TIID^Device 3 (NOV/DP-RAM)^Outputs^WorkOrderHmi} *)
	.NegToleranceEnabled AT %QX288.4 : BOOL;	(*  ~ {LinkedWith:TIID^Device 3 (NOV/DP-RAM)^Outputs^Var 278} *)
	.b16ConeModelSelected AT %QX288.5 : BOOL;
	.ProgramNoHmi AT %QB2276 : INT;	(*  ~ {LinkedWith:TIID^Device 3 (NOV/DP-RAM)^Outputs^PrgNo} *)
	.CountCodeHmi AT %QB2280 : STRING(80);	(*  ~ {LinkedWith:TIID^Device 3 (NOV/DP-RAM)^Outputs^CountCode} *)
	.CartonNoHmi AT %QB2362 : INT;	(*  ~ {LinkedWith:TIID^Device 3 (NOV/DP-RAM)^Outputs^CartonNo} *)
	.DefaultNetWeightHmi AT %QB2364 : REAL;	(*  ~ {LinkedWith:TIID^Device 3 (NOV/DP-RAM)^Outputs^DfltNetWt} *)
	.DefaultGrossWeightHmi AT %QB2368 : REAL;	(*  ~ {LinkedWith:TIID^Device 3 (NOV/DP-RAM)^Outputs^DfltGrossWt} *)
	.EmptyConeWt AT %QB3640 : REAL;	(*  ~ {LinkedWith:TIID^Device 3 (NOV/DP-RAM)^Outputs^EmptyConet} *)
	.BlendHmi AT %QB2372 : STRING(80);	(*  ~ {LinkedWith:TIID^Device 3 (NOV/DP-RAM)^Outputs^Blend} *)
	.ShadeHmi AT %QB2456 : STRING(80);	(*  ~ {LinkedWith:TIID^Device 3 (NOV/DP-RAM)^Outputs^Shade} *)
	.ConeTipHmi AT %QB2540 : STRING(80);	(*  ~ {LinkedWith:TIID^Device 3 (NOV/DP-RAM)^Outputs^ConeTip} *)
	.ConeNettHmi AT %QB2624 : STRING(80);	(*  ~ {LinkedWith:TIID^Device 3 (NOV/DP-RAM)^Outputs^ConeNetWt} *)
	.ConeLengthHmi AT %QB2708 : REAL;	(*  ~ {LinkedWith:TIID^Device 3 (NOV/DP-RAM)^Outputs^ConeLen} *)
	.Dom_ExpHmi AT %QB2712 : STRING(80);	(*  ~ {LinkedWith:TIID^Device 3 (NOV/DP-RAM)^Outputs^Dom} *)
	.PackTypeHmi AT %QB2796 : STRING(80);	(*  ~ {LinkedWith:TIID^Device 3 (NOV/DP-RAM)^Outputs^PackType} *)
	.ItemCodeHmi AT %QB2880 : STRING(80);	(*  ~ {LinkedWith:TIID^Device 3 (NOV/DP-RAM)^Outputs^ItemCode} *)
	.IssueDesp AT %QB2964 : STRING(80);	(*  ~ {LinkedWith:TIID^Device 3 (NOV/DP-RAM)^Outputs^IssueDes} *)
	.Location AT %QB3048 : STRING(80);	(*  ~ {LinkedWith:TIID^Device 3 (NOV/DP-RAM)^Outputs^Location} *)
	.Description AT %QB3132 : STRING(80);	(*  ~ {LinkedWith:TIID^Device 3 (NOV/DP-RAM)^Outputs^Description} *)
	.Remarks AT %QB3216 : STRING(80);	(*  ~ {LinkedWith:TIID^Device 3 (NOV/DP-RAM)^Outputs^Remarks} *)
	.Fyear AT %QB3300 : STRING(80);	(*  ~ {LinkedWith:TIID^Device 3 (NOV/DP-RAM)^Outputs^FYear} *)
	.AvgCount AT %QB3384 : STRING(80);	(*  ~ {LinkedWith:TIID^Device 3 (NOV/DP-RAM)^Outputs^Avg_Count} *)
	.TareWeight AT %QB3468 : REAL;	(*  ~ {LinkedWith:TIID^Device 3 (NOV/DP-RAM)^Outputs^TareWeight} *)
	.BarCode AT %QB3472 : STRING(80);	(*  ~ {LinkedWith:TIID^Device 3 (NOV/DP-RAM)^Outputs^Var 280} *)
	.WorkFlag AT %QB3556 : STRING(80);	(*  ~ {LinkedWith:TIID^Device 3 (NOV/DP-RAM)^Outputs^Var 279} *)
	.COMin_3_COMport_3 AT %IB56 : EL6inData22B;
	.COMout_3_COMport_3 AT %QB232 : EL6outData22B;
	.COMin_4_COMport_4 AT %IB80 : EL6inData22B;
	.COMout_4_COMport_4 AT %QB256 : EL6outData22B;
	.sGrosswt AT %QB280 : REAL;	(*  ~ {LinkedWith:TIID^Device 3 (NOV/DP-RAM)^Outputs^GrossWt} *)
	.sGrossTol AT %QB284 : REAL;	(*  ~ {LinkedWith:TIID^Device 3 (NOV/DP-RAM)^Outputs^GrossWtTol} *)
	.NegTolEnableHmi AT %QX2272.0 : BOOL;
	.NegTol1EnableHmi AT %QX2272.1 : BOOL;
	.NegTol2EnableHmi AT %QX2272.2 : BOOL;
	.NegTol3EnableHmi AT %QX2272.3 : BOOL;
	.NegTol4EnableHmi AT %QX2272.4 : BOOL;
	.NegTol5EnableHmi AT %QX2272.5 : BOOL;
	.PRGNO_DIS AT %QB292 : DINT;
	.COUNT_DIS AT %QB296 : STRING(80);
	.DETAILS_DIS AT %QB380 : STRING(80);
	.LOTNO_DIS AT %QB464 : STRING(80);
	.CARTONNO_DIS AT %QB548 : DINT;
	.DFLTNETWT_DIS AT %QB552 : REAL;
	.NETWTTOL_DIS AT %QB556 : REAL;
	.DFLTGROSSWT_DIS AT %QB560 : REAL;
	.GROSSWTTOL_DIS AT %QB564 : REAL;
	.NegTol_DIS AT %QB568 : REAL;
	.PRGNO AT %QB572 : DINT;
	.COUNT AT %QB576 : STRING(80);
	.DETAILS AT %QB660 : STRING(80);
	.LOTNO AT %QB744 : STRING(80);
	.CARTONNO AT %QB828 : DINT;
	.DFLTNETWT AT %QB832 : REAL;
	.NETWTTOL AT %QB836 : REAL;
	.DFLTGROSSWT AT %QB840 : REAL;
	.GROSSWTTOL AT %QB844 : REAL;
	.NegTol AT %QB848 : REAL;
	.PRGNO1 AT %QB852 : DINT;
	.COUNT1 AT %QB856 : STRING(80);
	.DETAILS1 AT %QB940 : STRING(80);
	.LOTNO1 AT %QB1024 : STRING(80);
	.CARTONNO1 AT %QB1108 : DINT;
	.DFLTNETWT1 AT %QB1112 : REAL;
	.NETWTTOL1 AT %QB1116 : REAL;
	.DFLTGROSSWT1 AT %QB1120 : REAL;
	.GROSSWTTOL1 AT %QB1124 : REAL;
	.NegTol1 AT %QB1128 : REAL;
	.PRGNO2 AT %QB1132 : DINT;
	.COUNT2 AT %QB1136 : STRING(80);
	.DETAILS2 AT %QB1220 : STRING(80);
	.LOTNO2 AT %QB1304 : STRING(80);
	.CARTONNO2 AT %QB1388 : DINT;
	.DFLTNETWT2 AT %QB1392 : REAL;
	.NETWTTOL2 AT %QB1396 : REAL;
	.DFLTGROSSWT2 AT %QB1400 : REAL;
	.GROSSWTTOL2 AT %QB1404 : REAL;
	.NegTol2 AT %QB1408 : REAL;
	.PRGNO3 AT %QB1412 : DINT;
	.COUNT3 AT %QB1416 : STRING(80);
	.DETAILS3 AT %QB1500 : STRING(80);
	.LOTNO3 AT %QB1584 : STRING(80);
	.CARTONNO3 AT %QB1668 : DINT;
	.DFLTNETWT3 AT %QB1672 : REAL;
	.NETWTTOL3 AT %QB1676 : REAL;
	.DFLTGROSSWT3 AT %QB1680 : REAL;
	.GROSSWTTOL3 AT %QB1684 : REAL;
	.NegTol3 AT %QB1688 : REAL;
	.PRGNO4 AT %QB1692 : DINT;
	.COUNT4 AT %QB1696 : STRING(80);
	.DETAILS4 AT %QB1780 : STRING(80);
	.LOTNO4 AT %QB1864 : STRING(80);
	.CARTONNO4 AT %QB1948 : DINT;
	.DFLTNETWT4 AT %QB1952 : REAL;
	.NETWTTOL4 AT %QB1956 : REAL;
	.DFLTGROSSWT4 AT %QB1960 : REAL;
	.GROSSWTTOL4 AT %QB1964 : REAL;
	.NegTol4 AT %QB1968 : REAL;
	.PRGNO5 AT %QB1972 : DINT;
	.COUNT5 AT %QB1976 : STRING(80);
	.DETAILS5 AT %QB2060 : STRING(80);
	.LOTNO5 AT %QB2144 : STRING(80);
	.CARTONNO5 AT %QB2228 : DINT;
	.DFLTNETWT5 AT %QB2232 : REAL;
	.NETWTTOL5 AT %QB2236 : REAL;
	.DFLTGROSSWT5 AT %QB2240 : REAL;
	.GROSSWTTOL5 AT %QB2244 : REAL;
	.NegTol5 AT %QB2248 : REAL;
	.PRG1RUNNING AT %QX2272.6 : BOOL;
	.PRG2RUNNING AT %QX2272.7 : BOOL;
	.PRG3RUNNING AT %QX2273.0 : BOOL;
	.PRG4RUNNING AT %QX2273.1 : BOOL;
	.PRG5RUNNING AT %QX2273.2 : BOOL;
	.SerialNo AT %QB2252 : DINT;
	.negativetolerance AT %QX2273.3 : BOOL;
	.DefaultNetWt AT %QB2256 : REAL;
	.NetWtTolRep AT %QB2260 : REAL;
	.DefaultGrossWt AT %QB2264 : REAL;	(*  ~ {LinkedWith:TIID^Device 3 (NOV/DP-RAM)^Outputs^Var 299} *)
	.GrossWtTolRep AT %QB2268 : REAL;
END_VAR

(* Global variable list: TwinCAT_Configuration_1 *)
(* Generated automatically by TwinCAT - (read only) *)
VAR_CONFIG
	.COMin_COMPort AT %IB8 : EL6inData22B;
	.COMOut_COMPort AT %QB4 : EL6outData22B;
	.COMin_2_COMport_2 AT %IB32 : EL6inData22B;
	.COMout_2_COMport_2 AT %QB28 : EL6outData22B;
END_VAR

(* Data type *)
TYPE Production_Data :
STRUCT

	S_No						:STRING;
	ConeType					:STRING;
	CartonNo					:STRING;
	LotNo						:STRING;
	SDateF						:STRING;
	NetWt						:STRING;
	WorkOrderNo				:STRING;
	DefaultNettWeight				:STRING;
	DefaultGrossWeight			:STRING;
	Blend						:STRING;
	Shade						:STRING;
	ConeTip						:STRING;
	ConeNettWeight				:STRING;
	ConeLength					:STRING;
	Dom_Exp					:STRING;
	PackType					:STRING;
	CountCode					:STRING;


END_STRUCT
END_TYPE

(* Data type *)
TYPE ProductionData_IndoPrint1 :
STRUCT
	SERIALNO			:STRING;
	SDATE				:STRING;
	NOOFCONE				:STRING;
	BAGNO				:STRING;
	COUNTCODE		:STRING;
	LOTNO				:STRING;
	DFLTNETWEIGHT	:STRING;
	DFLTGRSST		:STRING;
	ACTWT	:STRING;
	BLND	:STRING;
	SHD		:STRING;
	CONTIP				:STRING;
	CONNETWT	:STRING;
	CONLEN		:STRING;
	DOM	:STRING;
	ITEMCODE:STRING;
	PACKTYP	:STRING;
	WRKORNO	:STRING;
	COUNT	:STRING;
	TAREWEIGHTDET:STRING;
	WORKFLAGDET	:STRING;
	ISSUEDESPATCH	:STRING;
	REMARKSDET:STRING;
	LOCATIONDET	:STRING;
	DESCRIPTION	:STRING;
	FINYEAR	:STRING;
	AVERAGEGCOUNT	:STRING;
	BARCODE:STRING;
END_STRUCT
END_TYPE

(* Data type *)
TYPE ProductionData_PrintData :
STRUCT
	Print:STRING;
	PgNo:STRING;
	TotNoCones:STRING;
	CartNo:STRING;
	LotNo:STRING;
	DateTi:STRING;
	NetWt:STRING;
	WrkOrdNo:STRING;

	DfltNetWt:STRING;
	DfltGrsWt:STRING;
	Blnd:STRING;
	Shd:STRING;
	ConeTip:STRING;
	ConeNetWt:STRING;
	ConeLenght:STRING;
	Dom:STRING;
	Pack:STRING;
	CountCod:STRING;
END_STRUCT
END_TYPE

(* Data type *)
TYPE ST_CSV_Record :
STRUCT
	sName 	: T_MaxString 	:= '';
	nNumber	: UDINT 		:= 0;
	fPos		: LREAL 		:= 0.0;
	bOP		: BOOL 		:= FALSE;
	sDesc		: STRING(40)	:= '';
	data		: ARRAY[0..7] OF STRING;
END_STRUCT
END_TYPE

(* POU MAIN, ST *)
PROGRAM MAIN
VAR
	bTestBool: BOOL;
END_VAR
(*================== Model Selection Logic==========*)
IF bIAutoManual THEN bAutoModeOn:=TRUE; sAMcModeStatus:='Machine In Auto Mode'; bManualModeOn:=FALSE;

ELSIF NOT bIAutoManual THEN bManualModeOn:=TRUE;  sAMcModeStatus:='Machine In Manual Mode'; bAutoModeOn:=FALSE; END_IF

DATALOG_PRINT();
DATALOG_REPORT();
PARAMETER_SETTINGS();

One_Min_Conv();
FlimRollerUnit();
Auto();
UnitA_RowStopper();
UnitB_RowStopper();
Manual();
Outputs();
ConeFeedPiston();
ConeFeedConv();
Serial();
FwdPiston();

Wrapping_Unit();
Sealing_Unit();
Sealing_Conveyor();
WeightCalc();

INT_All();
Cylinder_Alarm();
ConeAllignAlarm();
ConeMiss_Alarm();
Common();

DataLog_1();

(*-===========Sealing Complete delay from Hmi==================*)

SealComDlyTemp:= REAL_TO_TIME(rSealCompDlyHmi * 1000);


(*==========Pause & Reume Logic====================*)


	IF bPauseHmi  OR bAPauseEnable THEN bAPauseSeq:=TRUE; END_IF
	IF bResumeHmi THEN bAPauseSeq:=FALSE; END_IF
END_PROGRAM

(* POU AutoMode/DATALOG_PRINT, ST *)
PROGRAM DATALOG_PRINT
VAR
	step: INT;
	bOpen: BOOL;
	FB_FileOpen1: FB_FileOpen;
	(*sPrintPath: STRING(80):= '\\PLC-PC\Reports\Print.csv';*)
	FB_FileWrite1: FB_FileWrite;
	FB_FileClose1: FB_FileClose;
	FB_FileDelete1: FB_FileDelete;

	TON_1: TON;
	bOpen1: BOOL;
	sHeadline: STRING;
	sData: STRING;
	ProductionData_PrintData: ProductionData_PrintData;

	PrintEnabled: BOOL;

	Timer_1: TON;
	Timer_2: TON;
	TON_2: TON;

	R_TRIGPrint: R_TRIG;
	TON_Opendly: TON;
	OpenError: INT;
	TON_writedly: TON;
	WriteError: INT;
	BlendPrint: STRING;
END_VAR
IF PrintEnableHmi THEN PrintEnabled:=TRUE;PrintValue:=1;ELSE PrintEnabled:=FALSE;PrintValue:=1;END_IF

BlendPrint:=CONCAT( BlendHmi , '%');
(*

		ProductionData_PrintData.Print						:=INT_TO_STRING( PrintValue );
		ProductionData_PrintData.ConeType1				:=(COUNT_DIS);
		ProductionData_PrintData.Blend1					:=(BLEND_DIS);
		ProductionData_PrintData.DefaultnetWt1				:=(NetwtPrint);
		ProductionData_PrintData.DefaultGrossWt1			:=(GrosswtPrint);
		ProductionData_PrintData.LotNo1					:=(LOTNO_DIS);
		ProductionData_PrintData.BagNo1					:=DINT_TO_STRING(CARTONNO_DIS);
		ProductionData_PrintData.Shade1					:=(SHADE_DIS);*)



ProductionData_PrintData.Print						:=INT_TO_STRING( PrintValue );
ProductionData_PrintData.PgNo						:=INT_TO_STRING( Pgm_NoHmi );
ProductionData_PrintData.TotNoCones						:=INT_TO_STRING( iATotalNoOfCones );
ProductionData_PrintData.CartNo						:=INT_TO_STRING(CartonNoHmi);
ProductionData_PrintData.LotNo						:=(iLotNoHmi);
ProductionData_PrintData.DateTi						:=(sDATEFinal);
ProductionData_PrintData.NetWt						:=REAL_TO_STRING(DefaultNetWeightHmi);
ProductionData_PrintData.WrkOrdNo						:=(iWorkOrderNoHmi);
ProductionData_PrintData.DfltNetWt						:=REAL_TO_STRING (DefaultNetWeightHmi);
ProductionData_PrintData.DfltGrsWt						:=REAL_TO_STRING(DefaultGrossWeightHmi);
ProductionData_PrintData.Blnd						:=(BlendPrint);
ProductionData_PrintData.Shd						:=(ShadeHmi );
ProductionData_PrintData.ConeTip						:=(ConeTipHmi);
ProductionData_PrintData.ConeNetWt						:=(ConeNettHmi);
ProductionData_PrintData.ConeLenght						:=REAL_TO_STRING (ConeLengthHmi);
ProductionData_PrintData.Dom						:=(Dom_ExpHmi);
ProductionData_PrintData.Pack						:=(PackTypeHmi);
ProductionData_PrintData.CountCod						:=(CountCodeHmi);


		(*	######## LOG PRODUCTION DATA		#####	*)

ProductionDataValues_Print:= CONCAT(ProductionData_PrintData.Print,',');
ProductionDataValues_Print:=	 CONCAT( ProductionDataValues_Print,ProductionData_PrintData.CountCod);
ProductionDataValues_Print:= CONCAT( ProductionDataValues_Print,',');
ProductionDataValues_Print:=	 CONCAT( ProductionDataValues_Print,ProductionData_PrintData.Blnd);
ProductionDataValues_Print:= CONCAT( ProductionDataValues_Print,',');
ProductionDataValues_Print:=	 CONCAT( ProductionDataValues_Print,ProductionData_PrintData.NetWt);
ProductionDataValues_Print:= CONCAT( ProductionDataValues_Print,',');
ProductionDataValues_Print:=	 CONCAT( ProductionDataValues_Print,ProductionData_PrintData.DfltGrsWt);
ProductionDataValues_Print:= CONCAT( ProductionDataValues_Print,',');
ProductionDataValues_Print:=	 CONCAT( ProductionDataValues_Print,ProductionData_PrintData.LotNo);
ProductionDataValues_Print:= CONCAT( ProductionDataValues_Print,',');
ProductionDataValues_Print:=	 CONCAT( ProductionDataValues_Print,ProductionData_PrintData.CartNo);
ProductionDataValues_Print:= CONCAT( ProductionDataValues_Print,',');
ProductionDataValues_Print:=	 CONCAT( ProductionDataValues_Print,ProductionData_PrintData.ConeTip);
ProductionDataValues_Print:= CONCAT( ProductionDataValues_Print,',');
ProductionDataValues_Print:=	 CONCAT( ProductionDataValues_Print,ProductionData_PrintData.Pack);
ProductionDataValues_Print:= CONCAT( ProductionDataValues_Print,',');
ProductionDataValues_Print:=	 CONCAT( ProductionDataValues_Print,ProductionData_PrintData.TotNoCones);
ProductionDataValues_Print:= CONCAT( ProductionDataValues_Print,',');
ProductionDataValues_Print:=	 CONCAT( ProductionDataValues_Print,ProductionData_PrintData.Shd);
ProductionDataValues_Print:= CONCAT( ProductionDataValues_Print,',');
ProductionDataValues_Print:=	 CONCAT( ProductionDataValues_Print,ProductionData_PrintData.ConeNetWt);
ProductionDataValues_Print:= CONCAT( ProductionDataValues_Print,',');
ProductionDataValues_Print:=	 CONCAT( ProductionDataValues_Print,ProductionData_PrintData.ConeLenght);
ProductionDataValues_Print:= CONCAT( ProductionDataValues_Print,'$0A');
(*ProductionDataValues_Print:=	 CONCAT( ProductionDataValues_Print,ProductionData_PrintData.WrkOrdNo);
ProductionDataValues_Print:= CONCAT( ProductionDataValues_Print,',');
ProductionDataValues_Print:=	 CONCAT( ProductionDataValues_Print,ProductionData_PrintData.DfltNetWt);
ProductionDataValues_Print:= CONCAT( ProductionDataValues_Print,',');
ProductionDataValues_Print:=	 CONCAT( ProductionDataValues_Print,ProductionData_PrintData.Dom);
ProductionDataValues_Print:= CONCAT( ProductionDataValues_Print,'$0A');*)




ProductionData_Print:= CONCAT( 'Print',',');
	ProductionData_Print:=	 CONCAT( ProductionData_Print,'Count');
ProductionData_Print:= CONCAT( ProductionData_Print,',');
	ProductionData_Print:=	 CONCAT( ProductionData_Print,'Blend');
ProductionData_Print:= CONCAT( ProductionData_Print,',');
	ProductionData_Print:=	 CONCAT( ProductionData_Print,'NetWt');
ProductionData_Print:= CONCAT( ProductionData_Print,',');
         ProductionData_Print:=	 CONCAT( ProductionData_Print,'GrossWt');
ProductionData_Print:= CONCAT( ProductionData_Print,',');
	ProductionData_Print:=	 CONCAT( ProductionData_Print,'LotNo');
ProductionData_Print:= CONCAT( ProductionData_Print,',');

	ProductionData_Print:=	 CONCAT( ProductionData_Print,'CartonNo');
ProductionData_Print:= CONCAT( ProductionData_Print,',');
	ProductionData_Print:=	 CONCAT( ProductionData_Print,'ConeTip');
ProductionData_Print:= CONCAT( ProductionData_Print,',');
	ProductionData_Print:=	 CONCAT( ProductionData_Print,'Pack');
ProductionData_Print:= CONCAT( ProductionData_Print,',');
	ProductionData_Print:=	 CONCAT( ProductionData_Print,'TotNoCone');
ProductionData_Print:= CONCAT( ProductionData_Print,',');

	ProductionData_Print:=	 CONCAT( ProductionData_Print,'Shade');
ProductionData_Print:= CONCAT( ProductionData_Print,',');
	ProductionData_Print:=	 CONCAT( ProductionData_Print,'ConeNetWt');
ProductionData_Print:= CONCAT( ProductionData_Print,',');

ProductionData_Print:=	 CONCAT( ProductionData_Print,'ConeLeng');
		ProductionData_Print:= CONCAT( ProductionData_Print,'$0A');
(*ProductionData_Print:=	 CONCAT( ProductionData_Print,'WorkOrdNo');
		ProductionData_Print:= CONCAT( ProductionData_Print,',');
ProductionData_Print:=	 CONCAT( ProductionData_Print,'DfltNtWt');
		ProductionData_Print:= CONCAT( ProductionData_Print,',');
ProductionData_Print:=	 CONCAT( ProductionData_Print,'Dom');
		ProductionData_Print:= CONCAT( ProductionData_Print,'$0A');*)








FB_FileOpen1(
	sNetId:='192.168.0.103.1.1' ,
	sPathName:= '\\Admin-PC\Reports\productiondata.csv' ,
	nMode:=FOPEN_MODEAPPEND ,
	ePath:=PATH_GENERIC ,
	bExecute:= ,
	tTimeout:=T#2s ,
	bBusy=> ,
	bError=> ,
	nErrId=> ,
	hFile=> );

FB_FileWrite1(
	sNetId:='192.168.0.103.1.1' ,
	hFile:=FB_FileOpen1.hFile ,
	pWriteBuff:=ADR(ProductionDataValues_Print_Com),
	cbWriteLen:=LEN(ProductionDataValues_Print_Com),
	bExecute:= ,
	tTimeout:=T#2s ,
	bBusy=> ,
	bError=> ,
	nErrId=> ,
	cbWrite=> );


FB_FileClose1(
	sNetId:='192.168.0.103.1.1' ,
	hFile:=FB_FileOpen1.hFile ,
	bExecute:= ,
	tTimeout:=T#2s ,
	bBusy=> ,
	bError=> ,
	nErrId=> );

FB_FileDelete1(
	sNetId:='192.168.0.103.1.1' ,
	sPathName:= '\\Admin-PC\Reports\productiondata.csv' ,
	ePath:=PATH_GENERIC ,
	bExecute:= ,
	tTimeout:=T#2s ,
	bBusy=> ,
	bError=> ,
	nErrId=> );

R_TRIGPrint(CLK:=CycleComplete OR CycleComplete1 , Q=> );

CASE step OF

0: IF R_TRIGPrint.Q THEN
	TON_2(IN:=FALSE);
	ReportSave:=TRUE;

	FB_FileOpen1.bExecute:=TRUE;
	IF NOT FB_FileOpen1.bBusy AND NOT FB_FileOpen1.bError AND FB_FileOpen1.hFile>0 THEN bOpen1:=FALSE; step:=step+1;END_IF
	END_IF


1:	IF NOT FB_FileOpen1.bBusy AND NOT FB_FileOpen1.bError AND FB_FileOpen1.hFile>0 THEN bOpen1:=FALSE; PrintOk:=FALSE;step:=step+1;END_IF

2:
	ProductionDataValues_Print_Com:=ProductionData_Print;
	FB_FileWrite1.bExecute:=TRUE;
	IF NOT FB_FileWrite1.bBusy AND NOT FB_FileWrite1.bError THEN step:=step+1;END_IF


3:	IF NOT FB_FileWrite1.bBusy AND NOT FB_FileWrite1.bError THEN FB_FileWrite1.bExecute:=FALSE; step:=step+1;END_IF

4:	ProductionDataValues_Print_Com:=ProductionDataValues_Print;
	FB_FileWrite1.bExecute:=TRUE;
	IF NOT FB_FileWrite1.bBusy AND NOT FB_FileWrite1.bError THEN step:=step+1;END_IF



5:	step:=step+1;


6:	IF NOT FB_FileWrite1.bBusy AND NOT FB_FileWrite1.bError THEN FB_FileWrite1.bExecute:=FALSE; step:=step+1;END_IF


7:	FB_FileClose1.bExecute:=TRUE;
	 IF NOT FB_FileClose1.bBusy AND NOT FB_FileClose1.bError THEN  step:=step+1;END_IF

8:	TON_1(IN:=TRUE , PT:=t#1s , Q=> , ET=> );
	IF TON_1.Q THEN step:=step+1;END_IF

9:	IF NOT FB_FileDelete1.bBusy AND NOT FB_FileDelete1.bError THEN
	TON_1(IN:=FALSE);
	(*FB_FileDelete1.bExecute:=TRUE;*)step:=step+1;END_IF

10:
	FB_FileOpen1.bExecute:=FALSE;
	FB_FileWrite1.bExecute:=FALSE;
	FB_FileClose1.bExecute:=FALSE;
	FB_FileDelete1.bExecute:=FALSE;
	bOpen:=FALSE;step:=step+1;

11:		TON_2(IN:=TRUE , PT:=t#10s , Q=> , ET=> );
	IF TON_2.Q THEN(* PrintOk:=TRUE;	*) step:=0;END_IF

END_CASE



CASE WriteError OF

0:	IF FB_FileWrite1.bError THEN FB_FileWrite1.bExecute:=FALSE;TON_writedly(IN:=FALSE);
	WriteError:=WriteError+1;END_IF

1:	TON_writedly(IN:=TRUE , PT:=t#2s , Q=> , ET=> );
	IF TON_writedly.Q THEN FB_FileWrite1.bExecute:=TRUE;WriteError:=WriteError+1;END_IF

2:	TON_writedly(IN:=FALSE);WriteError:=0;

END_CASE




CASE OpenError OF

0:	IF FB_FileOpen1.bError THEN FB_FileOpen1.bExecute:=FALSE;TON_Opendly(IN:=FALSE);
	OpenError:=OpenError+1;END_IF

1:	TON_Opendly(IN:=TRUE , PT:=t#2s , Q=> , ET=> );
	IF TON_Opendly.Q THEN FB_FileOpen1.bExecute:=TRUE;OpenError:=OpenError+1;END_IF

2:	TON_Opendly(IN:=FALSE);OpenError:=0;

END_CASE
END_PROGRAM

(* POU AutoMode/DATALOG_REPORT, ST *)
PROGRAM DATALOG_REPORT
VAR
	R_TRIG_IndoPrint: R_TRIG;
	FB_FileOpen_Indo: FB_FileOpen;
	FB_FileWrite_Indo: FB_FileWrite;
	FB_FileClose_Indo: FB_FileClose;
	FB_FileDelete_Indo: FB_FileDelete;
	IndoReport: INT;
	ReportHead1_Indo: BOOL;
	ST1_ProductionData: BOOL;
	ReportHead2_Indo: BOOL;
	ReportBot1_Indo: BOOL;
	stStation1_ProductionData: BOOL;
	ReportBot2_Indo: BOOL;
	testbit: BOOL;
	TON_Indo1: TON;
	TON_Indo2: TON;
	TON_Indo3: TON;
	TON_Indo4: TON;
	sOldDay: STRING;
	TON_Newdaydly: TON;
	TON_NEWDAY: TON;

	TON_NewdaydlyError: TON;
	WriteError: INT;
	TON_writedly: TON;
	OpenError: INT;
	TON_Opendly: TON;


	BarcodeNo: STRING;
	BarCode1: STRING;
	EmptyConeWtRep: REAL;
	EmptyConeWtRep1: REAL;
END_VAR
FB_FileOpen_Indo(
	sNetId:='192.168.0.103.1.1' ,
	sPathName:= ReportPath_Final_2,
	nMode:=FOPEN_MODEAPPEND ,
	ePath:=PATH_GENERIC ,
	bExecute:= ,
	tTimeout:=T#2s ,
	bBusy=> ,
	bError=> ,
	nErrId=> ,
	hFile=> );

FB_FileWrite_Indo(
	sNetId:='192.168.0.103.1.1' ,
	hFile:=FB_FileOpen_Indo.hFile ,
	pWriteBuff:=ADR(ProductionDataValues_IndoPrint_Com),
	cbWriteLen:=LEN(ProductionDataValues_IndoPrint_Com),
	bExecute:= ,
	tTimeout:=T#2s ,
	bBusy=> ,
	bError=> ,
	nErrId=> ,
	cbWrite=> );


FB_FileClose_Indo(
	sNetId:='192.168.0.103.1.1' ,
	hFile:=FB_FileOpen_Indo.hFile ,
	bExecute:= ,
	tTimeout:=T#2s ,
	bBusy=> ,
	bError=> ,
	nErrId=> );

FB_FileDelete_Indo(
	sNetId:='192.168.0.103.1.1' ,
	sPathName:=ReportPath_Final_2,
	ePath:=PATH_GENERIC ,
	bExecute:= ,
	tTimeout:=T#2s ,
	bBusy=> ,
	bError=> ,
	nErrId=> );

R_TRIG_IndoPrint(CLK:=( bANewDay OR testbit)  , Q=> );

CASE IndoReport OF
0:	  IF TON_NEWDAY.Q   THEN	sOldDay := sDay;TON_Newdaydly(IN:=TRUE , PT:=t#0.2s , Q=> , ET=> );
		IF TON_Newdaydly.Q THEN
		bANewDay:=FALSE;IndoReport:=1; SerialNoError:=1;FB_FileOpen_Indo.bExecute:=TRUE;END_IF END_IF

1:	TON_Newdaydly(IN:=FALSE);TON_NEWDAY(IN:=FALSE);
	IF NOT FB_FileOpen_Indo.bBusy AND NOT FB_FileOpen_Indo.bError AND FB_FileOpen_Indo.hFile>0 THEN ReportHead1_Indo:=TRUE;END_IF

	IF ReportHead1_Indo THEN
	ProductionData_IndoPrint:= CONCAT( 'DATE',',');
	ProductionData_IndoPrint:=	 CONCAT( ProductionData_IndoPrint,'DOM ');
		ProductionData_IndoPrint:= CONCAT( ProductionData_IndoPrint,',');
	ProductionData_IndoPrint:=	 CONCAT( ProductionData_IndoPrint,'BAG NO');
		ProductionData_IndoPrint:= CONCAT( ProductionData_IndoPrint,',');
	ProductionData_IndoPrint:=	 CONCAT( ProductionData_IndoPrint,' PACK');
		ProductionData_IndoPrint:= CONCAT( ProductionData_IndoPrint,',');
	ProductionData_IndoPrint:=	 CONCAT( ProductionData_IndoPrint,'ITEM CODE');
		ProductionData_IndoPrint:=CONCAT( ProductionData_IndoPrint,',');
	ProductionData_IndoPrint:=	 CONCAT( ProductionData_IndoPrint,'LOT NO');
		ProductionData_IndoPrint:=CONCAT( ProductionData_IndoPrint,',');
	ProductionData_IndoPrint:=	 CONCAT( ProductionData_IndoPrint,'COUNT');
		ProductionData_IndoPrint:=CONCAT( ProductionData_IndoPrint,',');

ProductionData_IndoPrint:=	 CONCAT( ProductionData_IndoPrint,'BLEND');
		ProductionData_IndoPrint:=CONCAT( ProductionData_IndoPrint,',');

ProductionData_IndoPrint:=	 CONCAT( ProductionData_IndoPrint,'SHDAE');
		ProductionData_IndoPrint:=CONCAT( ProductionData_IndoPrint,',');


ProductionData_IndoPrint:=	 CONCAT( ProductionData_IndoPrint,'CONES');
		ProductionData_IndoPrint:=CONCAT( ProductionData_IndoPrint,',');

ProductionData_IndoPrint:=	 CONCAT( ProductionData_IndoPrint,'NET WT');
		ProductionData_IndoPrint:=CONCAT( ProductionData_IndoPrint,',');

ProductionData_IndoPrint:=	 CONCAT( ProductionData_IndoPrint,'TARE WT');
		ProductionData_IndoPrint:=CONCAT( ProductionData_IndoPrint,',');


ProductionData_IndoPrint:=	 CONCAT( ProductionData_IndoPrint,'GR WT');
		ProductionData_IndoPrint:=CONCAT( ProductionData_IndoPrint,',');


ProductionData_IndoPrint:=	 CONCAT( ProductionData_IndoPrint,'CN WT');
		ProductionData_IndoPrint:=CONCAT( ProductionData_IndoPrint,',');

ProductionData_IndoPrint:=	 CONCAT( ProductionData_IndoPrint,'CN LEN');
		ProductionData_IndoPrint:=CONCAT( ProductionData_IndoPrint,',');

ProductionData_IndoPrint:=	 CONCAT( ProductionData_IndoPrint,'WORK ORDER');
		ProductionData_IndoPrint:=CONCAT( ProductionData_IndoPrint,',');

ProductionData_IndoPrint:=	 CONCAT( ProductionData_IndoPrint,'BAR CODE');
		ProductionData_IndoPrint:=CONCAT( ProductionData_IndoPrint,',');

	ProductionData_IndoPrint:=	 CONCAT( ProductionData_IndoPrint,'WORCP FLAG');
ProductionData_IndoPrint:=CONCAT( ProductionData_IndoPrint,',');
		(*ProductionData_IndoPrint:= CONCAT( ProductionData_IndoPrint,'$0A');*)
(*ProductionData_IndoPrint:=	 CONCAT( ProductionData_IndoPrint,'DFLT GROSS WT');
		ProductionData_IndoPrint:=CONCAT( ProductionData_IndoPrint,',');
ProductionData_IndoPrint:=	 CONCAT( ProductionData_IndoPrint,'ACT GROSS WT');
		ProductionData_IndoPrint:= CONCAT( ProductionData_IndoPrint,'$0A');
ProductionData_IndoPrint:=	 CONCAT( ProductionData_IndoPrint,'Cn9Wt');
		ProductionData_IndoPrint:=CONCAT( ProductionData_IndoPrint,',');
ProductionData_IndoPrint:=	 CONCAT( ProductionData_IndoPrint,'Cn10Wt');
		ProductionData_IndoPrint:=CONCAT( ProductionData_IndoPrint,',');
ProductionData_IndoPrint:=	 CONCAT( ProductionData_IndoPrint,'Cn11Wt');
		ProductionData_IndoPrint:=CONCAT( ProductionData_IndoPrint,',');
ProductionData_IndoPrint:=	 CONCAT( ProductionData_IndoPrint,'Cn12Wt');
	ProductionData_IndoPrint:=CONCAT( ProductionData_IndoPrint,',');*)
IndoReport:=2; END_IF

2:	PROCESSCOMPLETE:=FALSE;ReportHead1_Indo:=FALSE;ProductionDataValues_IndoPrint_Com:=ProductionData_IndoPrint;
	TON_Indo1(IN:=TRUE , PT:=t#5s , Q=> , ET=> );
	FB_FileWrite_Indo.bExecute:=TRUE;
	IF NOT FB_FileWrite_Indo.bBusy AND NOT FB_FileWrite_Indo.bError AND FB_FileWrite_Indo.hFile>0 AND TON_Indo1.Q THEN IndoReport:=IndoReport+1; END_IF

3:	ProductionDataValues_IndoPrint_Com:=ProductionData_IndoPrint;
	FB_FileWrite_Indo.bExecute:=TRUE;
	IF NOT FB_FileWrite_Indo.bBusy AND NOT FB_FileWrite_Indo.bError THEN IndoReport:=IndoReport+1; END_IF

4:	FB_FileWrite_Indo.bExecute:=FALSE;ProductionData_IndoPrint:='';IndoReport:=IndoReport+1;

5:	ReportHead2_Indo:=TRUE;
	IF ReportHead2_Indo THEN IndoReport:=IndoReport+1;END_IF

6:	ProductionData_IndoPrint:=	 CONCAT( ProductionData_IndoPrint,'ISSUE DESP');
		ProductionData_IndoPrint:=CONCAT( ProductionData_IndoPrint,',');
ProductionData_IndoPrint:=	 CONCAT( ProductionData_IndoPrint,'LOCATION');
		ProductionData_IndoPrint:=CONCAT( ProductionData_IndoPrint,',');
ProductionData_IndoPrint:=	 CONCAT( ProductionData_IndoPrint,'REMARKS');
		ProductionData_IndoPrint:=CONCAT( ProductionData_IndoPrint,',');
ProductionData_IndoPrint:=	 CONCAT( ProductionData_IndoPrint,'ITEM DESCR');
		ProductionData_IndoPrint:=CONCAT( ProductionData_IndoPrint,',');
ProductionData_IndoPrint:=	 CONCAT( ProductionData_IndoPrint,'CN TIP');
		ProductionData_IndoPrint:=CONCAT( ProductionData_IndoPrint,',');
ProductionData_IndoPrint:=	 CONCAT( ProductionData_IndoPrint,'ACT WT');
		ProductionData_IndoPrint:=CONCAT( ProductionData_IndoPrint,',');
ProductionData_IndoPrint:=	 CONCAT( ProductionData_IndoPrint,'FYEAR');
		ProductionData_IndoPrint:=CONCAT( ProductionData_IndoPrint,',');
(*ProductionData_IndoPrint:=	 CONCAT( ProductionData_IndoPrint,'Cn20Wt');
		ProductionData_IndoPrint:=CONCAT( ProductionData_IndoPrint,',');
ProductionData_IndoPrint:=	 CONCAT( ProductionData_IndoPrint,'Cn21Wt');
		ProductionData_IndoPrint:=CONCAT( ProductionData_IndoPrint,',');
ProductionData_IndoPrint:=	 CONCAT( ProductionData_IndoPrint,'Cn22Wt');
		ProductionData_IndoPrint:=CONCAT( ProductionData_IndoPrint,',');
ProductionData_IndoPrint:=	 CONCAT( ProductionData_IndoPrint,'Cn23Wt');
		ProductionData_IndoPrint:=CONCAT( ProductionData_IndoPrint,',');*)
	ProductionData_IndoPrint:=	 CONCAT( ProductionData_IndoPrint,'AVG COUNT');
ProductionData_IndoPrint:= CONCAT( ProductionData_IndoPrint,'$0A');
ReportHead2_Indo:=FALSE;
IndoReport:=IndoReport+1;

7:	ReportHead1_Indo:=FALSE;ProductionDataValues_IndoPrint_Com:=ProductionData_IndoPrint;
TON_Indo2(IN:=TRUE , PT:=t#5s , Q=> , ET=> );
	FB_FileWrite_Indo.bExecute:=TRUE;
	IF NOT FB_FileWrite_Indo.bBusy AND NOT FB_FileWrite_Indo.bError  AND TON_Indo2.Q THEN  IndoReport:=IndoReport+1; END_IF

8:	FB_FileWrite_Indo.bExecute:=FALSE;
	FB_FileClose_Indo.bExecute:=TRUE;
	 IF NOT FB_FileClose_Indo.bBusy AND NOT FB_FileClose_Indo.bError THEN FB_FileOpen_Indo.bExecute:=FALSE; IndoReport:=IndoReport+1;END_IF(*ProductionData_IndoPrint:='';*)

9:	FB_FileClose_Indo.bExecute:=FALSE;
	IF ReportSave OR testbit THEN

	FB_FileOpen_Indo.bExecute:=TRUE;
	IF NOT FB_FileOpen_Indo.bBusy AND NOT FB_FileOpen_Indo.bError AND FB_FileOpen_Indo.hFile>0 THEN  ReportBot1_Indo:=TRUE;END_IF

	IF ReportBot1_Indo THEN IndoReport:=IndoReport+1;END_IF END_IF

10:
ProductionData_IndoPrint2:= CONCAT(ProductionData_IndoPrint11.SDATE,',');
ProductionData_IndoPrint2:=	 CONCAT( ProductionData_IndoPrint2,ProductionData_IndoPrint11.DOM);
ProductionData_IndoPrint2:= CONCAT( ProductionData_IndoPrint2,',');
ProductionData_IndoPrint2:=	 CONCAT( ProductionData_IndoPrint2,ProductionData_IndoPrint11.BAGNO	);
ProductionData_IndoPrint2:= CONCAT( ProductionData_IndoPrint2,',');
ProductionData_IndoPrint2:=	 CONCAT( ProductionData_IndoPrint2,ProductionData_IndoPrint11.PACKTYP	);
ProductionData_IndoPrint2:= CONCAT( ProductionData_IndoPrint2,',');
ProductionData_IndoPrint2:=	 CONCAT( ProductionData_IndoPrint2,ProductionData_IndoPrint11.ITEMCODE);
ProductionData_IndoPrint2:= CONCAT( ProductionData_IndoPrint2,',');
ProductionData_IndoPrint2:=	 CONCAT( ProductionData_IndoPrint2,ProductionData_IndoPrint11.LOTNO);
ProductionData_IndoPrint2:= CONCAT( ProductionData_IndoPrint2,',');
ProductionData_IndoPrint2:=	 CONCAT( ProductionData_IndoPrint2,ProductionData_IndoPrint11.COUNT);
ProductionData_IndoPrint2:= CONCAT( ProductionData_IndoPrint2,',');

ProductionData_IndoPrint2:=	 CONCAT( ProductionData_IndoPrint2,ProductionData_IndoPrint11.BLND);
ProductionData_IndoPrint2:= CONCAT( ProductionData_IndoPrint2,',');

ProductionData_IndoPrint2:=	 CONCAT( ProductionData_IndoPrint2,ProductionData_IndoPrint11.SHD);
ProductionData_IndoPrint2:= CONCAT( ProductionData_IndoPrint2,',');
(*

ProductionData_IndoPrint2:=	 CONCAT( ProductionData_IndoPrint2,ProductionData_IndoPrint11.BLND);
ProductionData_IndoPrint2:= CONCAT( ProductionData_IndoPrint2,',');


ProductionData_IndoPrint2:=	 CONCAT( ProductionData_IndoPrint2,ProductionData_IndoPrint11.SHD);
ProductionData_IndoPrint2:= CONCAT( ProductionData_IndoPrint2,',');
*)

ProductionData_IndoPrint2:=	 CONCAT( ProductionData_IndoPrint2,ProductionData_IndoPrint11.NOOFCONE);
ProductionData_IndoPrint2:= CONCAT( ProductionData_IndoPrint2,',');


ProductionData_IndoPrint2:=	 CONCAT( ProductionData_IndoPrint2,ProductionData_IndoPrint11.DFLTNETWEIGHT);
ProductionData_IndoPrint2:= CONCAT( ProductionData_IndoPrint2,',');


ProductionData_IndoPrint2:=	 CONCAT( ProductionData_IndoPrint2,ProductionData_IndoPrint11.TAREWEIGHTDET);
ProductionData_IndoPrint2:= CONCAT( ProductionData_IndoPrint2,',');


ProductionData_IndoPrint2:=	 CONCAT( ProductionData_IndoPrint2,ProductionData_IndoPrint11.DFLTGRSST);
ProductionData_IndoPrint2:= CONCAT( ProductionData_IndoPrint2,',');


ProductionData_IndoPrint2:=	 CONCAT( ProductionData_IndoPrint2,ProductionData_IndoPrint11.CONNETWT);
ProductionData_IndoPrint2:= CONCAT( ProductionData_IndoPrint2,',');


ProductionData_IndoPrint2:=	 CONCAT( ProductionData_IndoPrint2,ProductionData_IndoPrint11.CONLEN);
ProductionData_IndoPrint2:= CONCAT( ProductionData_IndoPrint2,',');


ProductionData_IndoPrint2:=	 CONCAT( ProductionData_IndoPrint2,ProductionData_IndoPrint11.WRKORNO);
ProductionData_IndoPrint2:= CONCAT( ProductionData_IndoPrint2,',');
(*ProductionData_IndoPrint2:= CONCAT( ProductionData_IndoPrint2,'$0A');*)

ReportBot1_Indo:=FALSE;ReportSave:=FALSE;
IndoReport:=11;


11:	ProductionDataValues_IndoPrint_Com:=ProductionData_IndoPrint2;
	TON_Indo3(IN:=TRUE , PT:=t#5s , Q=> , ET=> );
	FB_FileWrite_Indo.bExecute:=TRUE;
	IF NOT FB_FileWrite_Indo.bBusy AND NOT FB_FileWrite_Indo.bError AND TON_Indo3.Q THEN IndoReport:=IndoReport+1; END_IF

12:	FB_FileWrite_Indo.bExecute:=FALSE;(*ProductionData_IndoPrint:='';*)IndoReport:=IndoReport+1;

13:	ReportBot2_Indo:=TRUE;
	IF ReportBot2_Indo THEN IndoReport:=IndoReport+1;END_IF

14:ProductionData_IndoPrint2:= CONCAT(ProductionData_IndoPrint11.BARCODE,',');
ProductionData_IndoPrint2:=	 CONCAT( ProductionData_IndoPrint2,ProductionData_IndoPrint11.WORKFLAGDET);
ProductionData_IndoPrint2:= CONCAT( ProductionData_IndoPrint2,',');
ProductionData_IndoPrint2:=	 CONCAT( ProductionData_IndoPrint2,ProductionData_IndoPrint11.ISSUEDESPATCH);
ProductionData_IndoPrint2:= CONCAT( ProductionData_IndoPrint2,',');
ProductionData_IndoPrint2:=	 CONCAT( ProductionData_IndoPrint2,ProductionData_IndoPrint11.LOCATIONDET);
ProductionData_IndoPrint2:= CONCAT( ProductionData_IndoPrint2,',');
ProductionData_IndoPrint2:=	 CONCAT( ProductionData_IndoPrint2,ProductionData_IndoPrint11.REMARKSDET);
ProductionData_IndoPrint2:= CONCAT( ProductionData_IndoPrint2,',');
ProductionData_IndoPrint2:=	 CONCAT( ProductionData_IndoPrint2,ProductionData_IndoPrint11.DESCRIPTION);
ProductionData_IndoPrint2:= CONCAT( ProductionData_IndoPrint2,',');
ProductionData_IndoPrint2:=	 CONCAT( ProductionData_IndoPrint2,ProductionData_IndoPrint11.CONTIP);
ProductionData_IndoPrint2:= CONCAT( ProductionData_IndoPrint2,',');
ProductionData_IndoPrint2:=	 CONCAT( ProductionData_IndoPrint2,ProductionData_IndoPrint11.ACTWT);
ProductionData_IndoPrint2:= CONCAT( ProductionData_IndoPrint2,',');
ProductionData_IndoPrint2:=	 CONCAT( ProductionData_IndoPrint2,ProductionData_IndoPrint11.FINYEAR);
ProductionData_IndoPrint2:= CONCAT( ProductionData_IndoPrint2,',');
(*ProductionData_IndoPrint2:=	 CONCAT( ProductionData_IndoPrint2,ProductionData_IndoPrint11.NetWt21);
ProductionData_IndoPrint2:= CONCAT( ProductionData_IndoPrint2,',');
ProductionData_IndoPrint2:=	 CONCAT( ProductionData_IndoPrint2,ProductionData_IndoPrint11.NetWt22);
ProductionData_IndoPrint2:= CONCAT( ProductionData_IndoPrint2,',');
ProductionData_IndoPrint2:=	 CONCAT( ProductionData_IndoPrint2,ProductionData_IndoPrint11.NetWt23);
ProductionData_IndoPrint2:= CONCAT( ProductionData_IndoPrint2,',');*)
ProductionData_IndoPrint2:=	 CONCAT( ProductionData_IndoPrint2,ProductionData_IndoPrint11.AVERAGEGCOUNT);
(*ProductionData_IndoPrint2:= CONCAT( ProductionData_IndoPrint2,',');*)
ProductionData_IndoPrint2:= CONCAT( ProductionData_IndoPrint2,'$0A');
ReportBot2_Indo:=FALSE;
IndoReport:=IndoReport+1;

15:ProductionDataValues_IndoPrint_Com:=ProductionData_IndoPrint2;
TON_Indo4(IN:=TRUE , PT:=t#5s , Q=> , ET=> );

	FB_FileWrite_Indo.bExecute:=TRUE; IndoReport:=IndoReport+1;
	(*IF NOT FB_FileWrite_Indo.bBusy AND NOT FB_FileWrite_Indo.bError AND TON_Indo4.Q  THEN IndoReport:=IndoReport+1;END_IF*)

16:	IF NOT FB_FileWrite_Indo.bBusy AND NOT FB_FileWrite_Indo.bError THEN FB_FileWrite_Indo.bExecute:=FALSE; IndoReport:=IndoReport+1;END_IF


17:	TON_Indo3(IN:=FALSE);TON_Indo4(IN:=FALSE);TON_Indo2(IN:=FALSE);TON_Indo1(IN:=FALSE);FB_FileWrite_Indo.bExecute:=FALSE;IndoReport:=IndoReport+1;

18:	FB_FileClose_Indo.bExecute:=TRUE;
	 IF NOT FB_FileClose_Indo.bBusy AND NOT FB_FileClose_Indo.bError THEN  IndoReport:=20;END_IF

19:	IF bANewDay THEN IndoReport:=IndoReport+1;
	ELSIF NOT bANewDay THEN FB_FileOpen_Indo.bExecute:=FALSE; IndoReport:=9;
END_IF

20:	FB_FileOpen_Indo.bExecute:=FALSE;SerialNo:=SerialNo+1;IndoReport:=9;

END_CASE



IF sDay <> sOldDay THEN bANewDay:=TRUE;IndoReport:=0; SerialNo:=0;END_IF
TON_NEWDAY(IN:=bANewDay , PT:=T#0.5s , Q=> , ET=> );




CASE WriteError OF

0:	IF FB_FileWrite_Indo.bError THEN FB_FileWrite_Indo.bExecute:=FALSE;TON_writedly(IN:=FALSE);
	WriteError:=WriteError+1;END_IF

1:	TON_writedly(IN:=TRUE , PT:=t#2s , Q=> , ET=> );
	IF TON_writedly.Q THEN FB_FileWrite_Indo.bExecute:=TRUE;WriteError:=WriteError+1;END_IF

2:	TON_writedly(IN:=FALSE);WriteError:=0;

END_CASE




CASE OpenError OF

0:	IF FB_FileOpen_Indo.bError THEN FB_FileOpen_Indo.bExecute:=FALSE;TON_Opendly(IN:=FALSE);
	OpenError:=OpenError+1;END_IF

1:	TON_Opendly(IN:=TRUE , PT:=t#2s , Q=> , ET=> );
	IF TON_Opendly.Q THEN FB_FileOpen_Indo.bExecute:=TRUE;OpenError:=OpenError+1;END_IF

2:	TON_Opendly(IN:=FALSE);OpenError:=0;

END_CASE

EmptyConeWtRep1:=(iATotalNoOfCones * EmptyConeWt);
EmptyConeWtRep:=(var_5  - EmptyConeWtRep1);

TareWeight:=(DefaultGrossWeightHmi - DefaultNetWeightHmi);


BarCode1:=CONCAT(STR1:=iLotNoHmi, STR2:='.');
BarCode:=CONCAT(STR1:=BarCode1, STR2:=(sBagNoRep));








	ProductionData_IndoPrint11.DOM	:= (Dom_ExpHmi);
	ProductionData_IndoPrint11.BAGNO	:=INT_TO_STRING(CartonNoHmi)(*CartonNoHmi*);
	ProductionData_IndoPrint11.PACKTYP	:=(PackTypeHmi);
	ProductionData_IndoPrint11.ITEMCODE	:=(ItemCodeHmi);
	ProductionData_IndoPrint11.LOTNO	:=(iLotNoHmi);
	ProductionData_IndoPrint11.COUNT	:=(CountCodeHmi);
	ProductionData_IndoPrint11.BLND	:=(BlendHmi);
	ProductionData_IndoPrint11.SHD	:=(ShadeHmi );
	ProductionData_IndoPrint11.NOOFCONE	:=INT_TO_STRING( iATotalNoOfCones );
	ProductionData_IndoPrint11.DFLTNETWEIGHT	:=REAL_TO_STRING(DefaultNetWeightHmi);
	ProductionData_IndoPrint11.TAREWEIGHTDET	:=REAL_TO_STRING(TareWeight);
	ProductionData_IndoPrint11.DFLTGRSST	:=REAL_TO_STRING(DefaultGrossWeightHmi);
	ProductionData_IndoPrint11.CONNETWT	:=(*REAL_TO_STRING*)(ConeNettHmi);
	ProductionData_IndoPrint11.CONLEN	:=REAL_TO_STRING (ConeLengthHmi);
	ProductionData_IndoPrint11.WRKORNO	:=(iWorkOrderNoHmi);
	ProductionData_IndoPrint11.BARCODE	:=(BarCode);
	ProductionData_IndoPrint11.WORKFLAGDET	:=(WorkFlag);
	ProductionData_IndoPrint11.ISSUEDESPATCH	:=(IssueDesp);
	ProductionData_IndoPrint11.LOCATIONDET	:=(Location);
	ProductionData_IndoPrint11.REMARKSDET	:=(Remarks);
	ProductionData_IndoPrint11.DESCRIPTION	:=(Description);
	ProductionData_IndoPrint11.CONTIP	:=(ConeTipHmi);
	ProductionData_IndoPrint11.ACTWT	:=REAL_TO_STRING(EmptyConeWtRep);
	ProductionData_IndoPrint11.FINYEAR	:=(Fyear);
	ProductionData_IndoPrint11.AVERAGEGCOUNT	:=(AvgCount);

		ProductionData_IndoPrint11.SERIALNO	:=INT_TO_STRING(Pgm_NoHmi);
		ProductionData_IndoPrint11.SDATE	:=(sDaateReport);
END_PROGRAM

(* POU AutoMode/PARAMETER_SETTINGS, ST *)
PROGRAM PARAMETER_SETTINGS
VAR
	R_TRIG_1: R_TRIG;

	PrintVar: INT;
	negativetolerance1: BOOL;
	negativetolerance2: BOOL;
	negativetolerance3: BOOL;
	negativetolerance4: BOOL;
	negativetolerance5: BOOL;
END_VAR
IF SAVE AND PRGNO=1 AND NegTolEnableHmi THEN NegTol1:=1;ELSIF SAVE AND PRGNO=1 AND NOT  NegTolEnableHmi THEN  NegTol1:=0;END_IF
IF SAVE AND PRGNO=2 AND NegTolEnableHmi THEN NegTol2:=1;ELSIF SAVE AND PRGNO=2 AND NOT NegTolEnableHmi THEN  NegTol2:=0;END_IF
IF SAVE AND PRGNO=3 AND NegTolEnableHmi THEN NegTol3:=1;ELSIF SAVE AND PRGNO=3 AND NOT NegTolEnableHmi THEN  NegTol3:=0;END_IF
IF SAVE AND PRGNO=4 AND NegTolEnableHmi THEN NegTol4:=1;ELSIF SAVE AND PRGNO=4 AND NOT NegTolEnableHmi THEN  NegTol4:=0;END_IF
IF SAVE AND PRGNO=5 AND NegTolEnableHmi THEN NegTol5:=1;ELSIF SAVE AND PRGNO=5 AND NOT NegTolEnableHmi THEN  NegTol5:=0;END_IF

IF SAVE AND PRGNO=1 THEN

	PRGNO1:=PRGNO;
	COUNT1:=COUNT;
	DETAILS1:=DETAILS;
	LOTNO1:=LOTNO;
	CARTONNO1:=CARTONNO;
	WORKORDERNO1:=WORKORDERNO;
	BLEND1:=BLEND;
	SHADE1:=SHADE;
	CONETIP1:=CONETIP;
	CONELENGTH1:=CONELENGTH;
	CONENETWT1:=CONENETWT;
	DFLTNETWT1:=DFLTNETWT;
	NETWTTOL1:=NETWTTOL;
	DFLTGROSSWT1:=DFLTGROSSWT;
	GROSSWTTOL1:=GROSSWTTOL;
	(*NegTol1:=NegTol;*)

ELSIF SAVE AND PRGNO=2 THEN

	PRGNO2:=PRGNO;
	COUNT2:=COUNT;
	DETAILS2:=DETAILS;
	LOTNO2:=LOTNO;
	CARTONNO2:=CARTONNO;
	WORKORDERNO2:=WORKORDERNO;
	BLEND2:=BLEND;
	SHADE2:=SHADE;
	CONETIP2:=CONETIP;
	CONELENGTH2:=CONELENGTH;
	CONENETWT2:=CONENETWT;
	DFLTNETWT2:=DFLTNETWT;
	NETWTTOL2:=NETWTTOL;
	DFLTGROSSWT2:=DFLTGROSSWT;
	GROSSWTTOL2:=GROSSWTTOL;
	(*NegTol2:=NegTol;*)

ELSIF SAVE AND PRGNO=3 THEN

	PRGNO3:=PRGNO;
	COUNT3:=COUNT;
	DETAILS3:=DETAILS;
	LOTNO3:=LOTNO;
	CARTONNO3:=CARTONNO;
	WORKORDERNO3:=WORKORDERNO;
	BLEND3:=BLEND;
	SHADE3:=SHADE;
	CONETIP3:=CONETIP;
	CONELENGTH3:=CONELENGTH;
	CONENETWT3:=CONENETWT;
	DFLTNETWT3:=DFLTNETWT;
	NETWTTOL3:=NETWTTOL;
	DFLTGROSSWT3:=DFLTGROSSWT;
	GROSSWTTOL3:=GROSSWTTOL;
	(*NegTol3:=NegTol;*)


ELSIF SAVE AND PRGNO=4 THEN

	PRGNO4:=PRGNO;
	COUNT4:=COUNT;
	DETAILS4:=DETAILS;
	LOTNO4:=LOTNO;
	CARTONNO4:=CARTONNO;
	WORKORDERNO4:=WORKORDERNO;
	BLEND4:=BLEND;
	SHADE4:=SHADE;
	CONETIP4:=CONETIP;
	CONELENGTH4:=CONELENGTH;
	CONENETWT4:=CONENETWT;
	DFLTNETWT4:=DFLTNETWT;
	NETWTTOL4:=NETWTTOL;
	DFLTGROSSWT4:=DFLTGROSSWT;
	GROSSWTTOL4:=GROSSWTTOL;
	(*NegTol4:=NegTol;*)

ELSIF SAVE AND PRGNO=5 THEN

	PRGNO5:=PRGNO;
	COUNT5:=COUNT;
	DETAILS5:=DETAILS;
	LOTNO5:=LOTNO;
	CARTONNO5:=CARTONNO;
	WORKORDERNO5:=WORKORDERNO;
	BLEND5:=BLEND;
	SHADE5:=SHADE;
	CONETIP5:=CONETIP;
	CONELENGTH5:=CONELENGTH;
	CONENETWT5:=CONENETWT;
	DFLTNETWT5:=DFLTNETWT;
	NETWTTOL5:=NETWTTOL;
	DFLTGROSSWT5:=DFLTGROSSWT;
	GROSSWTTOL5:=GROSSWTTOL;
	(*NegTol5:=NegTol;*)

ELSIF SAVE AND PRGNO=6 THEN

	PRGNO6:=PRGNO;
	COUNT6:=COUNT;
	DETAILS6:=DETAILS;
	LOTNO6:=LOTNO;
	CARTONNO6:=CARTONNO;
	WORKORDERNO6:=WORKORDERNO;
	BLEND6:=BLEND;
	SHADE6:=SHADE;
	CONETIP6:=CONETIP;
	CONELENGTH6:=CONELENGTH;
	CONENETWT6:=CONENETWT;
	DFLTNETWT6:=DFLTNETWT;
	NETWTTOL6:=NETWTTOL;
	DFLTGROSSWT6:=DFLTGROSSWT;
	GROSSWTTOL6:=GROSSWTTOL;


ELSIF SAVE AND PRGNO=7 THEN

	PRGNO7:=PRGNO;
	COUNT7:=COUNT;
	DETAILS7:=DETAILS;
	LOTNO7:=LOTNO;
	CARTONNO7:=CARTONNO;
	WORKORDERNO7:=WORKORDERNO;
	BLEND7:=BLEND;
	SHADE7:=SHADE;
	CONETIP7:=CONETIP;
	CONELENGTH7:=CONELENGTH;
	CONENETWT7:=CONENETWT;
	DFLTNETWT7:=DFLTNETWT;
	NETWTTOL7:=NETWTTOL;
	DFLTGROSSWT7:=DFLTGROSSWT;
	GROSSWTTOL7:=GROSSWTTOL;


ELSIF SAVE AND PRGNO=8 THEN

	PRGNO8:=PRGNO;
	COUNT8:=COUNT;
	DETAILS8:=DETAILS;
	LOTNO8:=LOTNO;
	CARTONNO8:=CARTONNO;
	WORKORDERNO8:=WORKORDERNO;
	BLEND8:=BLEND;
	SHADE8:=SHADE;
	CONETIP8:=CONETIP;
	CONELENGTH8:=CONELENGTH;
	CONENETWT8:=CONENETWT;
	DFLTNETWT8:=DFLTNETWT;
	NETWTTOL8:=NETWTTOL;
	DFLTGROSSWT8:=DFLTGROSSWT;
	GROSSWTTOL8:=GROSSWTTOL;


ELSIF SAVE AND PRGNO=9 THEN

	PRGNO9:=PRGNO;
	COUNT9:=COUNT;
	DETAILS9:=DETAILS;
	LOTNO9:=LOTNO;
	CARTONNO9:=CARTONNO;
	WORKORDERNO9 :=WORKORDERNO;
	BLEND9 :=BLEND;
	SHADE9 :=SHADE;
	CONETIP9 :=CONETIP;
	CONELENGTH9 :=CONELENGTH;
	CONENETWT9 :=CONENETWT;
	DFLTNETWT9 :=DFLTNETWT;
	NETWTTOL9 :=NETWTTOL;
	DFLTGROSSWT9 :=DFLTGROSSWT;
	GROSSWTTOL9 :=GROSSWTTOL;


ELSIF SAVE AND PRGNO=10 THEN

	PRGNO10:=PRGNO;
	COUNT10:=COUNT;
	DETAILS10:=DETAILS;
	LOTNO10:=LOTNO;
	CARTONNO10:=CARTONNO;
	WORKORDERNO10:=WORKORDERNO;
	BLEND10:=BLEND;
	SHADE10:=SHADE;
	CONETIP10:=CONETIP;
	CONELENGTH10:=CONELENGTH;
	CONENETWT10:=CONENETWT;
	DFLTNETWT10:=DFLTNETWT;
	NETWTTOL10:=NETWTTOL;
	DFLTGROSSWT10:=DFLTGROSSWT;
	GROSSWTTOL10:=GROSSWTTOL;

END_IF










IF LOAD AND PRGNO_LOAD=1 THEN

	PRGNO_DIS:=PRGNO1;
	COUNT_DIS:=COUNT1;
	DETAILS_DIS:=DETAILS1;
	LOTNO_DIS:=LOTNO1;
	CARTONNO_DIS:=CARTONNO1;
	WORKORDERNO_DIS:=WORKORDERNO1;
	BLEND_DIS:=BLEND1;
	SHADE_DIS:=SHADE1;
	CONETIP_DIS:=CONETIP1;
	CONELENGTH_DIS:=CONELENGTH1;
	CONENETWT_DIS:=CONENETWT1;
	DFLTNETWT_DIS:=DFLTNETWT1;
	NETWTTOL_DIS:=NETWTTOL1;
	DFLTGROSSWT_DIS:=DFLTGROSSWT1;
	GROSSWTTOL_DIS:=GROSSWTTOL1;
	NegTol_DIS:=NegTol1;
	PRG1RUNNING:=TRUE;
	PRG2RUNNING:=FALSE;
	PRG3RUNNING:=FALSE;
	PRG4RUNNING:=FALSE;
	PRG5RUNNING:=FALSE;
	PRG6RUNNING:=FALSE;
	PRG7RUNNING:=FALSE;
	PRG8RUNNING:=FALSE;
	PRG9RUNNING:=FALSE;
	PRG10RUNNING:=FALSE;

ELSIF LOAD AND PRGNO_LOAD=2 THEN

	PRGNO_DIS:=PRGNO2;
	COUNT_DIS:=COUNT2;
	DETAILS_DIS:=DETAILS2;
	LOTNO_DIS:=LOTNO2;
	CARTONNO_DIS:=CARTONNO2;
	WORKORDERNO_DIS:=WORKORDERNO2;
	BLEND_DIS:=BLEND2;
	SHADE_DIS:=SHADE2;
	CONETIP_DIS:=CONETIP2;
	CONELENGTH_DIS:=CONELENGTH2;
	CONENETWT_DIS:=CONENETWT2;
	DFLTNETWT_DIS:=DFLTNETWT2;
	NETWTTOL_DIS:=NETWTTOL2;
	DFLTGROSSWT_DIS:=DFLTGROSSWT2;
	GROSSWTTOL_DIS:=GROSSWTTOL2;
	NegTol_DIS:=NegTol2;
	PRG2RUNNING:=TRUE;
	PRG1RUNNING:=FALSE;
	PRG3RUNNING:=FALSE;
	PRG4RUNNING:=FALSE;
	PRG5RUNNING:=FALSE;
	PRG6RUNNING:=FALSE;
	PRG7RUNNING:=FALSE;
	PRG8RUNNING:=FALSE;
	PRG9RUNNING:=FALSE;
	PRG10RUNNING:=FALSE;

ELSIF LOAD AND PRGNO_LOAD=3 THEN

	PRGNO_DIS:=PRGNO3;
	COUNT_DIS:=COUNT3;
	DETAILS_DIS:=DETAILS3;
	LOTNO_DIS:=LOTNO3;
	CARTONNO_DIS:=CARTONNO3;
	WORKORDERNO_DIS:=WORKORDERNO3;
	BLEND_DIS:=BLEND3;
	SHADE_DIS:=SHADE3;
	CONETIP_DIS:=CONETIP3;
	CONELENGTH_DIS:=CONELENGTH3;
	CONENETWT_DIS:=CONENETWT3;
	DFLTNETWT_DIS:=DFLTNETWT3;
	NETWTTOL_DIS:=NETWTTOL3;
	DFLTGROSSWT_DIS:=DFLTGROSSWT3;
	GROSSWTTOL_DIS:=GROSSWTTOL3;
	NegTol_DIS:=NegTol3;
	PRG3RUNNING:=TRUE;
	PRG2RUNNING:=FALSE;
	PRG1RUNNING:=FALSE;
	PRG4RUNNING:=FALSE;
	PRG5RUNNING:=FALSE;
	PRG6RUNNING:=FALSE;
	PRG7RUNNING:=FALSE;
	PRG8RUNNING:=FALSE;
	PRG9RUNNING:=FALSE;
	PRG10RUNNING:=FALSE;


ELSIF LOAD AND PRGNO_LOAD=4 THEN

	PRGNO_DIS:=PRGNO4;
	COUNT_DIS:=COUNT4;
	DETAILS_DIS:=DETAILS4;
	LOTNO_DIS:=LOTNO4;
	CARTONNO_DIS:=CARTONNO4;
	WORKORDERNO_DIS:=WORKORDERNO4;
	BLEND_DIS:=BLEND4;
	SHADE_DIS:=SHADE4;
	CONETIP_DIS:=CONETIP4;
	CONELENGTH_DIS:=CONELENGTH4;
	CONENETWT_DIS:=CONENETWT4;
	DFLTNETWT_DIS:=DFLTNETWT4;
	NETWTTOL_DIS:=NETWTTOL4;
	DFLTGROSSWT_DIS:=DFLTGROSSWT4;
	GROSSWTTOL_DIS:=GROSSWTTOL4;
	NegTol_DIS:=NegTol4;
	PRG4RUNNING:=TRUE;
	PRG2RUNNING:=FALSE;
	PRG3RUNNING:=FALSE;
	PRG1RUNNING:=FALSE;
	PRG5RUNNING:=FALSE;
	PRG6RUNNING:=FALSE;
	PRG7RUNNING:=FALSE;
	PRG8RUNNING:=FALSE;
	PRG9RUNNING:=FALSE;
	PRG10RUNNING:=FALSE;


ELSIF LOAD AND PRGNO_LOAD=5 THEN

	PRGNO_DIS:=PRGNO5;
	COUNT_DIS:=COUNT5;
	DETAILS_DIS:=DETAILS5;
	LOTNO_DIS:=LOTNO5;
	CARTONNO_DIS:=CARTONNO5;
	WORKORDERNO_DIS:=WORKORDERNO5;
	BLEND_DIS:=BLEND5;
	SHADE_DIS:=SHADE5;
	CONETIP_DIS:=CONETIP5;
	CONELENGTH_DIS:=CONELENGTH5;
	CONENETWT_DIS:=CONENETWT5;
	DFLTNETWT_DIS:=DFLTNETWT5;
	NETWTTOL_DIS:=NETWTTOL5;
	DFLTGROSSWT_DIS:=DFLTGROSSWT5;
	GROSSWTTOL_DIS:=GROSSWTTOL5;
	NegTol_DIS:=NegTol5;
	PRG5RUNNING:=TRUE;
	PRG2RUNNING:=FALSE;
	PRG3RUNNING:=FALSE;
	PRG4RUNNING:=FALSE;
	PRG1RUNNING:=FALSE;
	PRG6RUNNING:=FALSE;
	PRG7RUNNING:=FALSE;
	PRG8RUNNING:=FALSE;
	PRG9RUNNING:=FALSE;
	PRG10RUNNING:=FALSE;

ELSIF LOAD AND PRGNO_LOAD=6 THEN

	PRGNO_DIS:=PRGNO6;
	COUNT_DIS:=COUNT6;
	DETAILS_DIS:=DETAILS6;
	LOTNO_DIS:=LOTNO6;
	CARTONNO_DIS:=CARTONNO6;
	WORKORDERNO_DIS:=WORKORDERNO6;
	BLEND_DIS:=BLEND6;
	SHADE_DIS:=SHADE6;
	CONETIP_DIS:=CONETIP6;
	CONELENGTH_DIS:=CONELENGTH6;
	CONENETWT_DIS:=CONENETWT6;
	DFLTNETWT_DIS:=DFLTNETWT6;
	NETWTTOL_DIS:=NETWTTOL6;
	DFLTGROSSWT_DIS:=DFLTGROSSWT6;
	GROSSWTTOL_DIS:=GROSSWTTOL6;
	PRG6RUNNING:=TRUE;
	PRG2RUNNING:=FALSE;
	PRG3RUNNING:=FALSE;
	PRG4RUNNING:=FALSE;
	PRG5RUNNING:=FALSE;
	PRG1RUNNING:=FALSE;
	PRG7RUNNING:=FALSE;
	PRG8RUNNING:=FALSE;
	PRG9RUNNING:=FALSE;
	PRG10RUNNING:=FALSE;

ELSIF LOAD AND PRGNO_LOAD=7 THEN

	PRGNO_DIS:=PRGNO7;
	COUNT_DIS:=COUNT7;
	DETAILS_DIS:=DETAILS7;
	LOTNO_DIS:=LOTNO7;
	CARTONNO_DIS:=CARTONNO7;
	WORKORDERNO_DIS:=WORKORDERNO7;
	BLEND_DIS:=BLEND7;
	SHADE_DIS:=SHADE7;
	CONETIP_DIS:=CONETIP7;
	CONELENGTH_DIS:=CONELENGTH7;
	CONENETWT_DIS:=CONENETWT7;
	DFLTNETWT_DIS:=DFLTNETWT7;
	NETWTTOL_DIS:=NETWTTOL7;
	DFLTGROSSWT_DIS:=DFLTGROSSWT7;
	GROSSWTTOL_DIS:=GROSSWTTOL7;
	PRG7RUNNING:=TRUE;
	PRG2RUNNING:=FALSE;
	PRG3RUNNING:=FALSE;
	PRG4RUNNING:=FALSE;
	PRG5RUNNING:=FALSE;
	PRG6RUNNING:=FALSE;
	PRG1RUNNING:=FALSE;
	PRG8RUNNING:=FALSE;
	PRG9RUNNING:=FALSE;
	PRG10RUNNING:=FALSE;


ELSIF LOAD AND PRGNO_LOAD=8 THEN

	PRGNO_DIS:=PRGNO8;
	COUNT_DIS:=COUNT8;
	DETAILS_DIS:=DETAILS8;
	LOTNO_DIS:=LOTNO8;
	CARTONNO_DIS:=CARTONNO8;
	WORKORDERNO_DIS:=WORKORDERNO8;
	BLEND_DIS:=BLEND8;
	SHADE_DIS:=SHADE8;
	CONETIP_DIS:=CONETIP8;
	CONELENGTH_DIS:=CONELENGTH8;
	CONENETWT_DIS:=CONENETWT8;
	DFLTNETWT_DIS:=DFLTNETWT8;
	NETWTTOL_DIS:=NETWTTOL8;
	DFLTGROSSWT_DIS:=DFLTGROSSWT8;
	GROSSWTTOL_DIS:=GROSSWTTOL8;
	PRG8RUNNING:=TRUE;
	PRG2RUNNING:=FALSE;
	PRG3RUNNING:=FALSE;
	PRG4RUNNING:=FALSE;
	PRG5RUNNING:=FALSE;
	PRG6RUNNING:=FALSE;
	PRG7RUNNING:=FALSE;
	PRG1RUNNING:=FALSE;
	PRG9RUNNING:=FALSE;
	PRG10RUNNING:=FALSE;


ELSIF LOAD AND PRGNO_LOAD=9 THEN

	PRGNO_DIS:=PRGNO9;
	COUNT_DIS:=COUNT9;
	DETAILS_DIS:=DETAILS9;
	LOTNO_DIS:=LOTNO9;
	CARTONNO_DIS:=CARTONNO9;
	WORKORDERNO_DIS:=WORKORDERNO9;
	BLEND_DIS:=BLEND9;
	SHADE_DIS:=SHADE9;
	CONETIP_DIS:=CONETIP9;
	CONELENGTH_DIS:=CONELENGTH9;
	CONENETWT_DIS:=CONENETWT9;
	DFLTNETWT_DIS:=DFLTNETWT9;
	NETWTTOL_DIS:=NETWTTOL9;
	DFLTGROSSWT_DIS:=DFLTGROSSWT9;
	GROSSWTTOL_DIS:=GROSSWTTOL9;
	PRG9RUNNING:=TRUE;
	PRG2RUNNING:=FALSE;
	PRG3RUNNING:=FALSE;
	PRG4RUNNING:=FALSE;
	PRG5RUNNING:=FALSE;
	PRG6RUNNING:=FALSE;
	PRG7RUNNING:=FALSE;
	PRG8RUNNING:=FALSE;
	PRG1RUNNING:=FALSE;
	PRG10RUNNING:=FALSE;


ELSIF LOAD AND PRGNO_LOAD=10 THEN

	PRGNO_DIS:=PRGNO10;
	COUNT_DIS:=COUNT10;
	DETAILS_DIS:=DETAILS10;
	LOTNO_DIS:=LOTNO10;
	CARTONNO_DIS:=CARTONNO10;
	WORKORDERNO_DIS:=WORKORDERNO10;
	BLEND_DIS:=BLEND10;
	SHADE_DIS:=SHADE10;
	CONETIP_DIS:=CONETIP10;
	CONELENGTH_DIS:=CONELENGTH10;
	CONENETWT_DIS:=CONENETWT10;
	DFLTNETWT_DIS:=DFLTNETWT10;
	NETWTTOL_DIS:=NETWTTOL10;
	DFLTGROSSWT_DIS:=DFLTGROSSWT10;
	GROSSWTTOL_DIS:=GROSSWTTOL10;
	PRG10RUNNING:=TRUE;
	PRG2RUNNING:=FALSE;
	PRG3RUNNING:=FALSE;
	PRG4RUNNING:=FALSE;
	PRG5RUNNING:=FALSE;
	PRG6RUNNING:=FALSE;
	PRG7RUNNING:=FALSE;
	PRG8RUNNING:=FALSE;
	PRG9RUNNING:=FALSE;
	PRG1RUNNING:=FALSE;

END_IF


IF PRG1RUNNING AND NegTol1=1 THEN negativetolerance1:=TRUE; ELSE negativetolerance1:=FALSE;END_IF

IF PRG2RUNNING AND NegTol2=1 THEN negativetolerance2:=TRUE; ELSE negativetolerance2:=FALSE;END_IF

IF PRG3RUNNING AND NegTol3=1 THEN negativetolerance3:=TRUE; ELSE negativetolerance3:=FALSE;END_IF

IF PRG4RUNNING AND NegTol4=1 THEN negativetolerance4:=TRUE; ELSE negativetolerance4:=FALSE;END_IF

IF PRG5RUNNING AND NegTol5=1 THEN negativetolerance5:=TRUE; ELSE negativetolerance5:=FALSE;END_IF

IF PRG1RUNNING AND negativetolerance1 THEN negativetolerance:=TRUE;
ELSIF PRG2RUNNING AND negativetolerance2 THEN negativetolerance:=TRUE;
ELSIF PRG3RUNNING AND negativetolerance3 THEN negativetolerance:=TRUE;
ELSIF PRG4RUNNING AND negativetolerance4 THEN negativetolerance:=TRUE;
ELSIF PRG5RUNNING AND negativetolerance5 THEN negativetolerance:=TRUE;END_IF
IF LOAD THEN negativetolerance:=FALSE;END_IF

R_TRIG_1(CLK:=(PROCESSCOMPLETE) , Q=> );


IF R_TRIG_1.Q THEN
CartonNoHmi:=CartonNoHmi+1;
(*CARTONNO_DIS:=CARTONNO_DIS+1;*)


END_IF

IF PRGNO_LOAD=3 AND R_TRIG_1.Q THEN CARTONNO3:=CARTONNO_DIS;
ELSIF PRGNO_LOAD=2 AND R_TRIG_1.Q THEN CARTONNO2:=CARTONNO_DIS;
ELSIF PRGNO_LOAD=1 AND R_TRIG_1.Q THEN CARTONNO1:=CARTONNO_DIS;
ELSIF PRGNO_LOAD=4 AND R_TRIG_1.Q THEN CARTONNO4:=CARTONNO_DIS;
ELSIF PRGNO_LOAD=5 AND R_TRIG_1.Q THEN CARTONNO5:=CARTONNO_DIS;
ELSIF PRGNO_LOAD=6 AND R_TRIG_1.Q THEN CARTONNO6:=CARTONNO_DIS;
ELSIF PRGNO_LOAD=7 AND R_TRIG_1.Q THEN CARTONNO7:=CARTONNO_DIS;
ELSIF PRGNO_LOAD=8 AND R_TRIG_1.Q THEN CARTONNO8:=CARTONNO_DIS;
ELSIF PRGNO_LOAD=9 AND R_TRIG_1.Q THEN CARTONNO9:=CARTONNO_DIS;
ELSIF PRGNO_LOAD=10 AND R_TRIG_1.Q THEN CARTONNO10:=CARTONNO_DIS;
END_IF

DefaultNetWt :=DFLTNETWT_DIS;
NetWtTolRep:=	NETWTTOL_DIS;
DefaultGrossWt:=	DFLTGROSSWT_DIS;
GrossWtTolRep:=	GROSSWTTOL_DIS;
END_PROGRAM

(* POU AutoMode/One_Min_Conv, ST *)
PROGRAM One_Min_Conv
VAR
	TON_5: TON;
	TON_6: TON;
	rGrossWtTolMin: REAL;
	rGrossWtTolMax: REAL;
	bGrossWieghtOkTemp: BOOL;
	bQAGrossWtPiston1: BOOL;
	bcheck: BOOL;

	TEST1: BOOL;
	TEST2: BOOL;
	tGrossWtEndSenDly: TON;
	CylErrChkBit: BOOL;
END_VAR
IF NOT  bIEmergency   OR bStopHmi  OR  bAutoModeOff  OR bIMCStop THEN
One_Min_Conv_1:=0;
bQGross_Roller_On:=FALSE; TON_5(IN:=FALSE); TON_6(IN:=FALSE);
END_IF
rGrossWtTolMax:= (sGrosswt + sGrossTol);

rGrossWtTolMin:= (sGrosswt - sGrossTol);


CASE One_Min_Conv_1 OF


	0:	IF bAutoModeOn AND bIGross_Crossing_Input  AND bAMcStartInAuto   AND NOT bAPauseSeq THEN
		bQGross_Roller_On:=TRUE; TON_5(IN:=FALSE);
		One_Min_Conv_1:=One_Min_Conv_1+1; END_IF

	1:	TON_5(IN:=TRUE , PT:=t#10S , Q=> , ET=> );
		IF  bIGross_Weight_Stop   AND NOT bAPauseSeq AND NOT  TON_5.Q THEN  One_Min_Conv_1:=One_Min_Conv_1+1;
		ELSE
		 IF  TON_5.Q THEN bcheck:=TRUE;  bQGross_Roller_On:=FALSE;  One_Min_Conv_1:=0;
		END_IF
		END_IF

	2:	IF bAutoModeOn AND bIGross_Weight_Stop   AND NOT bAPauseSeq THEN
		tGrossWtEndSenDly(IN:= FALSE);
		bQGross_Roller_On:=FALSE; bQGross_Cylinder_On:=TRUE;
		(*tGrossWtEndSenDly(IN:= TRUE, PT:=t#5s , Q=> , ET=> ); *)
		CylErrChkBit:=TRUE;
		One_Min_Conv_1:=One_Min_Conv_1+1; END_IF

	3:	IF bIGross_Cyl_End THEN 	CylErrChkBit:=FALSE; One_Min_Conv_1:=One_Min_Conv_1+1;
		ELSIF NOT bIGross_Cyl_End AND tGrossWtEndSenDly.Q THEN
		bGrossWtCylEndSenError:=TRUE;
		SGrossWtCylEndSenErrMsg:='Gross weight Cyl End Sensor Error';
		One_Min_Conv_1:=13;
		END_IF

	4:	TON_6(IN:=TRUE , PT:=t#9.5S , Q=> , ET=> );
		 IF  TON_6.Q THEN One_Min_Conv_1:=One_Min_Conv_1+1;  END_IF

	5:	IF  rGrossWeight >=rGrossWtTolMin  AND  rGrossWeight  <= rGrossWtTolMax  THEN
		bGrossWieghtOkTemp:=TRUE; rGrossWeighToReport:=rGrossWeight ;  bGrossWieghtNokTemp:=FALSE;
		One_Min_Conv_1:=One_Min_Conv_1+1;
		ELSIF  rGrossWeight  >  rGrossWtTolMax THEN
		bGrossWieghtNokTemp:=TRUE; bGrossWieghtOkTemp:=FALSE;
		One_Min_Conv_1:=One_Min_Conv_1+2;
		ELSIF   rGrossWeight  < rGrossWtTolMin   THEN
		bGrossWieghtNokTemp:=TRUE; bGrossWieghtOkTemp:=FALSE;
		One_Min_Conv_1:=One_Min_Conv_1+2;
		END_IF

	6:	IF bGrossWieghtOkTemp (*AND TEST1*)  THEN bGrossWieghtOk:=TRUE; bQAGrossWieghtOkIndi:=TRUE; One_Min_Conv_1:=One_Min_Conv_1+2;  TON_6(IN:=FALSE);  END_IF

	7:	IF bGrossWieghtNokTemp  (*AND TEST2 *)THEN bGrossWieghtNOk:=TRUE;
		SGrossWtNokMsg:='Gross Weight is Less OR more';
		bReadGWieght:=FALSE; One_Min_Conv_1:=One_Min_Conv_1+2;   TON_6(IN:=FALSE); END_IF


	8:	IF bGrossWieghtOk (*  AND NOT bGrossWieghtNok *) AND bAutoModeOn  AND NOT bAPauseSeq THEN
		 bQGross_Cylinder_On:=FALSE; bReadGWieght:=FALSE; bGrossWieghtOkTemp:=FALSE;
		bQAGrossWieghtOkIndi:=FALSE;   (*====== Modified for  Gross  Weight   bypass  ==============*)
		bACyclePass:=TRUE;
		GrossWtReedSwBit:=TRUE;
		One_Min_Conv_1:=One_Min_Conv_1+2;
		 END_IF

	9:	IF bErrorReset THEN  bGrossWieghtNOk:=FALSE;
		SGrossWtNokMsg:='';
		One_Min_Conv_1:=4; END_IF

	10:	IF bIGross_Cyl_Home  AND NOT bAGrossWtHomeSenRsError THEN GrossWtReedSwBit:=FALSE ; bQGross_Roller_On:=TRUE;  One_Min_Conv_1:=One_Min_Conv_1+1;END_IF

	11:	bACyclePass:=FALSE;One_Min_Conv_1:=One_Min_Conv_1+1;

	12:	IF bAutoModeOn AND NOT  bIGross_Weight_Stop   AND NOT bAPauseSeq THEN
		 One_Min_Conv_1:=0;  bQGross_Roller_On:=FALSE; END_IF

	13:	IF bErrorReset AND bIGross_Cyl_End THEN
		CylErrChkBit:=FALSE;
		bGrossWtCylEndSenError:=FALSE;
		tGrossWtEndSenDly(IN:= FALSE);
		SGrossWtCylEndSenErrMsg:='';
		One_Min_Conv_1:=2;
		ELSIF NOT bIGross_Cyl_End AND bErrorReset THEN
		CylErrChkBit:=FALSE;
		bGrossWtCylEndSenError:=FALSE;
		tGrossWtEndSenDly(IN:= FALSE);
		SGrossWtCylEndSenErrMsg:='';
		One_Min_Conv_1:=2;
		END_IF
END_CASE





IF CylErrChkBit THEN tGrossWtEndSenDly(IN:= TRUE, PT:=t#5s , Q=> , ET=> );
END_IF
END_PROGRAM

(* POU AutoMode/FlimRollerUnit, ST *)
PROGRAM FlimRollerUnit
VAR
	step: INT;
	bQAFilmRollerMotor1OnAuto: BOOL;
	bQAFilmRollerMotor2OnAuto: BOOL;
	bQAFilmRollerMotor3OnAuto: BOOL;
END_VAR
bQAFilmRollerMotor1:= ( bQAFilmRollerMotor1OnAuto );

bQAFilmRollerMotor2:= ( bQAFilmRollerMotor2OnAuto );

bQAFilmRollerMotor3:=( bQAFilmRollerMotor3OnAuto );





		IF NOT 	bIWrappingFilmTensionPlate_1  THEN
		bQAFilmRollerMotor1OnAuto:=TRUE;
		ELSE
		bQAFilmRollerMotor1OnAuto:=FALSE;
		END_IF


		IF NOT	bIWrappingFilmTensionPlate_2   THEN
		bQAFilmRollerMotor2OnAuto:=TRUE;
		ELSE
		bQAFilmRollerMotor2OnAuto:=FALSE;
		END_IF



		IF NOT	bIWrappingFilmTensionPlate_3    THEN
		bQAFilmRollerMotor3OnAuto:=TRUE;
		ELSE
		bQAFilmRollerMotor3OnAuto:=FALSE;
		END_IF
END_PROGRAM

(* POU AutoMode/Auto, ST *)
PROGRAM Auto
VAR
	Timer1: TON;
	Timer2: TON;
	bAmber: BOOL;
	bAGreen: BOOL;
	bARed: BOOL;
	bABuzzertest: BOOL;
	bABuzzertemp: BOOL;
	bAmberTemp: BOOL;
	bAmberbit1: BOOL;
END_VAR
	IF bAutoModeOn AND bIMCStart THEN bAMcStartInAuto:=TRUE; bAStop:=FALSE;  END_IF

	IF NOT bIEmergency OR  bIMCStop OR bStopHmi   THEN bAMcStartInAuto:=FALSE; END_IF


IF bAutoModeOff THEN bAMcStartInAuto:=FALSE; END_IF




(*=================Model Selection Logic===============*)

IF b12ConeModelHmi AND NOT  b18ConeModelHmi AND NOT  b24ConeModelHmi AND NOT b32ConeModelHmi AND NOT bInterlockInitial_2 THEN
b12ConeModelSelected:=TRUE; b16ConeModelSelected:=FALSE; b18ConeModelSelected:=FALSE; b24ConeModelSelected:=FALSE; b32ConeModelSelected:=FALSE;  END_IF

IF NOT  b12ConeModelHmi AND   b18ConeModelHmi AND NOT  b24ConeModelHmi AND NOT b32ConeModelHmi AND NOT bInterlockInitial_2 THEN
b18ConeModelSelected:=TRUE;   b16ConeModelSelected:=FALSE; b12ConeModelSelected:=FALSE; b24ConeModelSelected:=FALSE; b32ConeModelSelected:=FALSE;   END_IF

IF  NOT b12ConeModelHmi AND NOT  b18ConeModelHmi AND   b24ConeModelHmi AND NOT b32ConeModelHmi AND NOT bInterlockInitial_2 THEN
 b24ConeModelSelected:=TRUE; b16ConeModelSelected:=FALSE;  b18ConeModelSelected:=FALSE; b12ConeModelSelected:=FALSE; b32ConeModelSelected:=FALSE;    END_IF

IF  NOT b12ConeModelHmi AND NOT  b18ConeModelHmi AND NOT  b24ConeModelHmi AND  b32ConeModelHmi AND NOT bInterlockInitial_2  THEN
b32ConeModelSelected:=TRUE;  b18ConeModelSelected:=FALSE; b24ConeModelSelected:=FALSE; b12ConeModelSelected:=FALSE;    END_IF

IF  b16ConeModelHmi AND NOT b12ConeModelHmi AND NOT  b18ConeModelHmi AND NOT  b24ConeModelHmi AND  NOT b32ConeModelHmi  AND NOT bInterlockInitial_2 THEN
 b16ConeModelSelected:=TRUE;b32ConeModelSelected:=FALSE;  b18ConeModelSelected:=FALSE; b24ConeModelSelected:=FALSE; b12ConeModelSelected:=FALSE;    END_IF


IF b12ConeModelSelected THEN iATotalNoOfCones:=12;
ELSIF b16ConeModelSelected THEN iATotalNoOfCones:=16;
ELSIF  b18ConeModelSelected THEN iATotalNoOfCones:=18;
ELSIF  b24ConeModelSelected THEN iATotalNoOfCones:=24;
ELSIF  b32ConeModelSelected THEN iATotalNoOfCones:=32;
END_IF


Timer1(IN:=(bAInializeStarted AND NOT Timer2.Q   ) ,  PT:=t#0.5s , Q=> , ET=>, );
Timer2(IN:= Timer1.Q, PT:=t#0.5s , Q=> , ET=> );

IF bIMCStart THEN bAGreen:=TRUE; END_IF

IF Timer1.Q    AND NOT  bAError   AND NOT bAStop AND NOT bAPauseSeq THEN bAmber :=TRUE; bAGreen:=FALSE;  ELSE  bAmber:=FALSE; END_IF

IF Timer1.Q OR bAMcRunninig   OR bAMcReady AND NOT bAError AND NOT bAStop  THEN bAGreen :=TRUE;   ELSE  bAGreen:=FALSE; END_IF

IF Timer1.Q OR bAStop OR  bStopHmi THEN bARed :=TRUE; (*bAGreen:=FALSE;*)  bABuzzer:=FALSE; ELSE  bARed:=FALSE; END_IF
IF  bAPauseSeq THEN bAmberbit1 :=TRUE; bAGreen:=FALSE; ELSE bAmberbit1 :=FALSE; END_IF
IF Timer1.Q  AND NOT bAPauseSeq THEN  bAmber :=TRUE;  ELSE  bAmber :=FALSE;END_IF
IF bAError THEN  bAmberbit2:=TRUE;bAGreen:=FALSE;ELSE bAmberbit2 :=FALSE;END_IF

bQAAmber:=bAmber  OR bABuzzer OR bAmberbit1 OR bAmberbit2 ;
bQAGreen:= bAGreen;
bQARed:=bARed;
 bQABuzzer:= bABuzzer;

IF NOT  bIEmergency OR bStopHmi  OR bAutoModeOff OR bIMCStop  THEN bARed :=TRUE; bAGreen:=FALSE; bAmber:=FALSE; bAMcRunninig:=FALSE; END_IF
END_PROGRAM

(* POU AutoMode/UnitA_RowStopper, ST *)
PROGRAM UnitA_RowStopper
VAR
	step: INT;

	iSensorOnVal:UINT;
	CTU_1Enable: BOOL;
	R_TRIG_1: F_TRIG;
	CTU_2: CTU;
	R_TRIG_2: R_TRIG;
	tRowStopperRevDly1: TON;
	UnitAConeCrossCount: CTU;
	test: BOOL;
	bStopRetUnitA: BOOL;
	RowStopperMotorStopDly: TON;
	bRetUnitAStarttemp: BOOL;
	bAUnitAWeighOktemp: BOOL;
	RowStopperEndRSErrorDly: TON;
	bStartTemp1: BOOL;
	UnitAOverTemp: BOOL;
	RowStopperEndSenErr: BOOL;
	interLockStep: INT;
	UnitACompleteCheckCountCv: INT;
	bEnableBit1: BOOL;
	UnitAConeCross: CTU;
	Testtimer: TON;
	bAUnitBConeCrossingOff_2: BOOL;
	step3: INT;
	TON_7: TON;
	R_TRIG_4: R_TRIG;
	timer3: TON;

	SenSelect_1: SenSelect;
	iAConeCrossCount: INT;
	bQAUnitA_RowStopperMotorFwd2: BOOL;
	bQAUnitA_RowStopperMotorFwd1: BOOL;
	bQAUnitA_RowStopperMotorRev1: BOOL;
	sRetreivalAStatus: STRING;
	bRetUnitARst: BOOL;
	iAConeCrossCounttemp: INT;
	GetDLy: TON;
	bCheckSensor: BOOL;
	tConeChkDly: TON;
	bUnitAConeMiss:BOOL ;
	iAConeCrossPVal: INT;
	tConeCrossDly: TON;
	step2: INT;
	F_TRIG_5: F_TRIG;
	TON_6: TON;
	bAUnitBConeCrossing_1: BOOL;
	bAUnitBConeCrossingOff: BOOL;
	step4: INT;
	TON_8: TON;
	bAUnitAConeCrossing_1: BOOL;
	TON_9: TON;
	bAUnitAConeCrossingOff: BOOL;
	TON_10: TON;
	F_TRIG_3: F_TRIG;
	CountAtLimitBNok: BOOL;
	CountCheckdly: TON;
	UnitAConeCompChkCount: CTU;
	tRowStopperMidDly1: TON;
	tUnitACountDelay1: TON;
	TEnableCounter: BOOL;
	CompleteTestbitA: BOOL;
	bCounterLockUnitA: BOOL;
	bStartUnitaCompCount: BOOL;
END_VAR
UnitASenSelet:=iSensorOnVal;

(*=============Checking the No of sensors sensed================*)

IF bCheckSensor THEN
SenSelect_1(
		bVarIn1:=bIUnitAConeDetection1 ,
		bVarIn2:= bIUnitAConeDetection2,
		bVarIn3:= bIUnitAConeDetection3,
		bVarIn4:= bIUnitAConeDetection4,
		ByteResult=>iSensorOnVal );


END_IF

IF iSensorOnVal=15 THEN iAConeCrossCount:=4;
		ELSIF  iSensorOnVal=14 THEN iAConeCrossCount:=3;
		ELSIF  iSensorOnVal=13 THEN iAConeCrossCount:=3;
		ELSIF  iSensorOnVal=12 THEN iAConeCrossCount:=2;
		ELSIF  iSensorOnVal=11 THEN iAConeCrossCount:=3;
		ELSIF  iSensorOnVal=10 THEN iAConeCrossCount:=2;
		ELSIF  iSensorOnVal=9 THEN iAConeCrossCount:=2;
		ELSIF  iSensorOnVal=8 THEN iAConeCrossCount:=1;
		ELSIF  iSensorOnVal=7 THEN iAConeCrossCount:=3;
		ELSIF  iSensorOnVal=6 THEN iAConeCrossCount:=2;
		ELSIF  iSensorOnVal=5 THEN iAConeCrossCount:=2;
		ELSIF  iSensorOnVal=4 THEN iAConeCrossCount:=1;
		ELSIF  iSensorOnVal=3 THEN iAConeCrossCount:=2;
		ELSIF  iSensorOnVal=2 THEN iAConeCrossCount:=1;
		ELSIF  iSensorOnVal=1 THEN iAConeCrossCount:=1;
		END_IF





bQAUnitA_RowStopperMotorForward1:=( bQAUnitA_RowStopperMotorFwd1 OR bQAUnitA_RowStopperMotorFwd2 );

bQAUnitA_RowStopperMotorReverse1:= ( bQAUnitA_RowStopperMotorRev1 OR bRetUnitARst );

CASE step OF

	0:	IF bAutoModeOn AND bAUnitAWeighOk  AND bRetUnitAStart   AND NOT bAInializeStarted  AND NOT bIntialAckBit  AND bInterlockInitial_2 THEN
		CTU_2.RESET:=TRUE;

		step:=step+1;
		END_IF

	1:	step:=step+1;

	2:	IF bAutoModeOn(* AND bIUnitA_LiftPistonHome  *)THEN
		step:=step+1;


		END_IF

	3:	UnitAConeCompChkCount.RESET:=FALSE;
		TestTimer(IN:=FALSE);
		step:=step+1;

	4:	IF bAutoModeOn    AND NOT bUnitBRowStopperStarted  AND NOT UnitB_RowStopper.ConeInCompleteB  (*ConeInCompleteTestbitB*)
		AND NOT bAPauseSeq  AND NOT ConeInCompleteA   AND bInterlockInitial_2 THEN
		bQAUnitA_RowStopperMotorFwd1:=TRUE;
		UnitAConeCrossCount.RESET:=TRUE;
		bAUnitAWeighOk:=FALSE;

		bUnitARowStopperStarted:=TRUE;
		sRetreivalAStatus:= 'Running';

		 step:=step+1;
		END_IF

	5:	RowStopperMotorStopDly(In:=FALSE);
		 step:=step+1;

	6:	IF bIUnitAConeDetection1 OR  bIUnitAConeDetection2 OR  bIUnitAConeDetection3 OR   bIUnitAConeDetection4  THEN

		step:=step+1;
		ELSIF NOT bIUnitAConedetection1 AND NOT  bIUnitAConedetection2 AND NOT  bIUnitAConedetection3 AND NOT bIUnitAConeDetection4 AND  bIUnitA_RowStopperEnd THEN

		step:=15;
		END_IF

	7:	CompleteTestbitA:=FALSE;
		RowStopperMotorStopDly( IN:=TRUE , PT:=T#0.4s , Q=> , ET=> );
		IF RowStopperMotorStopDly.Q THEN  UnitAConeCrossCount.RESET:=FALSE;  step:=step+1; END_IF


	8:	bStartUnitaCompCount:=TRUE;
		bQAUnitA_RowStopperMotorFwd1:=FALSE;
		GetDLy(IN:=FALSE);
		tRowStopperRevDly1(IN:=FALSE);
		step:=step+1;

	9:	 IF  NOT   bAPauseSeq THEN  bCheckSensor:=TRUE;

		step:=step+1;

		END_IF


	10:	GetDLy(IN:=TRUE , PT:=t#0.4s , Q=> , ET=> );
		 IF GetDLy.Q THEN bCheckSensor:=FALSE;   step:=step+1;
		END_IF





	11:	IF UnitAConeCrossCount.CV=iAConeCrossCount  THEN
		RowStopperMotorStopDly(In:=FALSE);
		GetDLy(IN:=FALSE);
		step:=step+1;
		ELSIF UnitAConeCrossCount.CV <> iAConeCrossCount  THEN
		tConeChkDly(IN:=TRUE , PT:=t#5s , Q=> , ET=> );

	 (*	IF tConeChkDly.Q THEN bUnitAConeMiss:=TRUE; ELSE bUnitAConeMiss:=FALSE ;  END_IF *)
		END_IF

	12:	IF NOT bAPauseSeq THEN step:=step+1;
		END_IF

	13:	IF bAutoModeOn   THEN
		 UnitAConeCrossCount.RESET:=TRUE;
		step:=step+1;
		END_IF

	14:	UnitAConeCrossCount.RESET:=FALSE; step:=step+1;


	15: 	IF bAutoModeOn AND bIUnitA_RowStopperEnd THEN
		bQAUnitA_RowStopperMotorFwd1:=FALSE;
		tRowStopperRevDly1(IN:=FALSE);
		 step:=step+1;
		ELSIF  bAutoModeOn AND NOT  bIUnitA_RowStopperEnd THEN
		 step:=4;
		END_IF

	16:	step:=step+1;

	17:	tRowStopperRevDly1(IN:=TRUE , PT:=t#1.5s , Q=> , ET=> );
		IF tRowStopperRevDly1.Q THEN step:=step+1; END_IF

	18:	 step:=step+1;


	19:	IF bAutoModeOn   THEN
		bQAUnitA_RowStopperMotorRev1:=TRUE;
		PROCESSCOMPLETE:=TRUE;
		step:=step+1;
		END_IF

	20:	IF bAutoModeOn AND bIUnitA_RowStopperMiddle   THEN
		PROCESSCOMPLETE:=FALSE;
		tUnitACountDelay1(IN:=FALSE);
		tRowStopperMidDly1(IN:=TRUE , PT:=t#0.2s , Q=> , ET=> );
		IF tRowStopperMidDly1.Q THEN  step:=step+1;
		END_IF
		END_IF


	21:	tUnitACountDelay1(IN:=TRUE , PT:=t#5s , Q=> , ET=> );
		IF tUnitACountDelay1.Q THEN
		step:=step+1;
		END_IF




	22:	IF bAutoModeOn  AND UnitAConeCompChkCount.CV>=iATotalNoOfCones   THEN
		bUnitARowStopperStarted:=FALSE;
		UnitAConeCompChkCount.RESET:=TRUE;
		bStartUnitaCompCount:=FALSE;
		TestTimer(IN:=FALSE);
                  	step:=step+1;
		ELSIF  bAutoModeOn  AND UnitAConeCompChkCount.CV < iATotalNoOfCones  THEN
		TestTimer(IN:=FALSE);
		 ConeInCompleteA:=TRUE;
	(*	ConeInCompletetest:=TRUE; *)
		bStartUnitaCompCount:=FALSE;
		step:=step+1;

		END_IF


	23:	IF bAutoModeOn AND bIUnitA_RowStopperHome   AND ConeInCompleteA  THEN
		bQAUnitA_RowStopperMotorRev1:=FALSE;
		tRowStopperMidDly1(IN:=FALSE);
		sRetreivalAStatus:= 'IDLE';
		step:=0;
		ELSIF  bAutoModeOn AND bIUnitA_RowStopperHome   AND NOT ConeInCompleteA  THEN
		bQAUnitA_RowStopperMotorRev1:=FALSE;
		tRowStopperMidDly1(IN:=FALSE);
		sRetreivalAStatus:= 'IDLE';
		step:=0;
		END_IF

END_CASE

(***Incomplete Reset**)

IF  bAutoModeOn AND ConeInCompleteA   THEN
TEnableCounter:=TRUE;
ELSE
TEnableCounter:=FALSE;
END_IF



IF  bAutoModeOn AND ConeInCompleteA   AND   UnitAConeCompChkCount.CV >= iATotalNoOfCones THEN
TestTimer(IN:=TRUE , PT:=t#5s , Q=> , ET=> );
CycleComplete:=TRUE;
END_IF


IF TestTimer.Q THEN
CycleComplete:=FALSE;
UnitAConeCompChkCount.RESET:=TRUE;
bUnitARowStopperStarted:=FALSE;
ConeInCompleteA :=FALSE;
TestTimer(IN:=FALSE);
END_IF
(*

IF  bAutoModeOn AND UnitAConeCompChkCount.CV >= iATotalNoOfCones THEN
TEnableCounter:=FALSE;
tUnitACountDelay1(IN:=FALSE);
ConeInComplete:=FALSE;

END_IF

IF   bAutoModeOn  AND UnitAConeCompChkCount.CV >=iATotalNoOfCones   AND( bUnitARowStopperStarted OR ConeInCompletetest) THEN
CompleteTestbitA:=TRUE;
bStartUnitaCompCount:=FALSE;
UnitAConeCompChkCount.RESET:=TRUE;
ConeInCompletetest:=FALSE;
ELSE
UnitAConeCompChkCount.RESET:=FALSE;
END_IF
*)
UnitAConeCrossCount(
	CU:= bAUnitAConeCrossing_1  (*   R_TRIG_1.Q*) ,
	RESET:= ,
	PV:=12,
	Q=> ,
	CV=> );



UnitAConeCompChkCount(
	CU:=  bAUnitBConeCrossing_1 ,
	RESET:= ,
	PV:=iATotalNoOfCones,
	Q=> ,
	CV=> );
UnitAConeCountHMI:=UnitAConeCompChkCount.CV;

(*=======For Retrival A Limit Switch======*)
(*
LimitSwitchBCount(
	CU:=  bAUnitBConeCrossing_1,
	RESET:= ,
	PV:=iATotalNoOfCones,
	Q=> ,
	CV=> );
*)

IF UnitAConeCompChkCount.CV >=  iATotalNoOfCones AND bIUnitA_RowStopperHome  AND NOT bQAUnitA_RowStopperMotorRev1 AND NOT ConeInCompleteA  THEN tConeCrossDly(IN:=TRUE , PT:=t#0.5s , Q=> , ET=> );  END_IF
(*
IF LimitSwitchBCount.CV< iATotalNoOfCones AND bUnitARowStopperStarted THEN  CountAtLimitBNok:=TRUE;ELSE CountAtLimitBNok:=FALSE;  (*CountCheckdly(IN:=TRUE , PT:=t#5s , Q=> , ET=> )*); END_IF*)

IF tConeCrossDly.Q THEN bUnitARowStopperStarted:=FALSE; UnitAConeCompChkCount.RESET:=TRUE; step:=0;  tConeCrossDly(IN:=FALSE); ELSE  UnitAConeCompChkCount.RESET:=FALSE; END_IF

(*
ELSE
UnitAConeCompChkCount.RESET:=FALSE; *)



(*===============Stop Sequence===========*)


IF NOT bIEmergency  OR  bStopHmi  OR bAutoModeOff  OR bIMCStop   THEN bStopRetUnitA:=TRUE; END_IF


IF bStopRetUnitA (*AND NOT  bIUnitA_RowStopperHome *) THEN
step:=0;
step2:=0;
step4:=0;
bAUnitAWeighOk:=FALSE;
bQAUnitA_RowStopperMotorFwd1:=FALSE;
bUnitARowStopperStarted:=FALSE;
UnitAConeCrossCount.RESET:=FALSE;
bQAUnitA_RowStopperMotorFwd2:=FALSE;
UnitAConeCompChkCount.RESET:=TRUE;
bQAUnitA_RowStopperMotorRev1:=FALSE;
bRetUnitARst:=TRUE;
bAUnitAConeCrossing_1:=FALSE;
bAUnitBConeCrossing_1:=FALSE;
END_IF

IF bIUnitA_RowStopperHome THEN
bRetUnitARst:=FALSE;
  UnitAConeCompChkCount.RESET:=FALSE;
bStopRetUnitA:=FALSE;
END_IF

(*
(*=============for Pause Operation bypass to Feeding Conveyor==================*)

IF UnitAConeCrossCount.CV >= 1 AND bPauseHmi AND  UnitAConeCrossCount.CV=iAConeCrossCount THEN bPauseExtend:=TRUE; ELSE  bPauseExtend:=FALSE;  END_IF


*)



(*IF NOT CompleteTestbitA THEN  *)
CASE step2 OF

	0:	IF   (bStartUnitaCompCount  (*bUnitARowStopperStarted  *) OR  TEnableCounter  ) THEN
		F_TRIG_3(CLK:=bIUnitBConeCrossing , Q=> );
		IF F_TRIG_3.Q THEN TON_6(IN:= FALSE); step2:=step2+1; END_IF END_IF


	1:	TON_6(IN:= FALSE);
		TON_9(IN:= FALSE);
		step2:=step2+1;


	2:	 bAUnitBConeCrossing_1 :=TRUE;
		 step2:=Step2+1;

	3:	 step2:=step2+1;

	4: 	TON_6(IN:=  TRUE  , PT:=t#100ms,Q=> , ET=> );
		IF TON_6.Q THEN bAUnitBConeCrossing_1:=FALSE;   step2:=step2+1; END_IF


	5:	 step2:=step2+1;

	6:	IF   bIUnitBConeCrossing THEN
		TON_9(IN:=  TRUE  , PT:=t#50ms,Q=> , ET=>);
		IF TON_9.Q THEN TON_6(IN:= FALSE);  step2:=step2+1; END_IF END_IF


	7:	 step2:=step2+1;

	8:	 step2:=step2+1;

	9:	 step2:=step2+1;

	10:	TON_9(IN:= FALSE);
		step2:=0;


END_CASE
(*END_IF *)


CASE step4 OF

	0:	IF bUnitARowStopperStarted THEN
		F_TRIG_5(CLK:=bIUnitAConeCrossing , Q=> );
		IF F_TRIG_5.Q THEN TON_8(IN:= FALSE); step4:=step4+1; END_IF END_IF


	1:	TON_8(IN:= FALSE);
		TON_10(IN:= FALSE);
		step4:=step4+1;


	2:	 bAUnitAConeCrossing_1 :=TRUE;
		 step4:=step4+1;

	3:	 step4:=step4+1;

	4: 	TON_8(IN:=  TRUE  , PT:=t#100ms,Q=> , ET=> );
		IF TON_8.Q THEN  bAUnitAConeCrossing_1:=FALSE;  step4:=step4+1; END_IF


	5:	 step4:=step4+1;

	6:	IF   bIUnitAConeCrossing THEN
		TON_10(IN:=  TRUE  , PT:=t#50ms,Q=> , ET=>);
		IF TON_10.Q THEN TON_8(IN:= FALSE);  step4:=step4+1; END_IF END_IF


	7:	 step4:=step4+1;;

	8:	 step4:=step4+1;

	9:	 step4:=step4+1;

	10:	TON_8(IN:= FALSE);
		step4:=0;


END_CASE


IF bRetUnitAStart THEN step4:=0; step2:=0 ; END_IF
END_PROGRAM

(* POU FunctionBlocks/SenSelect, ST *)
FUNCTION_BLOCK SenSelect
VAR_INPUT


	bVarIn1: BOOL;
	bVarIn2: BOOL;
	bVarIn3: BOOL;
	bVarIn4: BOOL;
END_VAR
VAR_OUTPUT


	ByteResult: USINT;
END_VAR
VAR

END_VAR
ByteResult.0:=bVarIn1;
ByteResult.1:=bVarIn2;
ByteResult.2:=bVarIn3;
ByteResult.3:=bVarIn4;

ByteResult;
END_FUNCTION_BLOCK

(* POU AutoMode/UnitB_RowStopper, ST *)
PROGRAM UnitB_RowStopper
VAR
	step: INT;
	bAUnitAWeighOk: BOOL;
	CTU_1: CTU;
	CTU_1Enable: BOOL;
	R_TRIG_1: R_TRIG;
	R_TRIG_2: F_TRIG;
	bQAUnitA_RowStopperMotorFwd1: BOOL;
	bQAUnitA_RowStopperMotorFwd2: BOOL;
	tRowStopperRevDly1: TON;
	bQAUnitA_RowStopperMotorRev1: BOOL;
	CTU_2: CTU;
	UnitBConeCount: CTU;
	CTU_1EnableUnitB: BOOL;
	temp1: BOOL;
	bStopRetUnitB: BOOL;
	bRetUnitBRst: BOOL;
	RowStopperMotorStopDly: TON;
	F_TRIG_3: F_TRIG;
	UnitBCompleteCheckCount:CTU;
	UnitBOverTemp: BOOL;
	bStartTemp1: BOOL;
	R_TRIG_5: R_TRIG;
	test: BOOL;
	bStopTemp2: BOOL;
	CTU_2CV: INT;
	CTU_test: CTU;
	R_TRIG_test: R_TRIG;
	InterLockStep: INT;

	CTU_2Enable: BOOL;
	timer1: TON;
	UnitBCompleteCheckCountCV: INT;
	Ctu_2_Rst: BOOL;
	F_TRIG_1: F_TRIG;
	bRestBit: BOOL;
	bResetBit: BOOL;
	R_TRIG_6: R_TRIG;
	timer2: TON;
	UnitBConeCrossCount: CTU;
	bQAUnitB_RowStopperMotorFwd1: BOOL;
	sRetreivalBStatus: STRING;
	GetDLy: TON;
	bCheckSensor: BOOL;
	iAConeCrossCount: INT;
	bQAUnitB_RowStopperMotorRev1: BOOL;
	iSensorOnVal: USINT;
	SenSelect_2: SenSelect;
	tConeChkDly: TON;
	bConeMiss: BOOL;
	tConeCrossDly: TON;
	UnitBConeCompChkCount: CTU;
	iAConeCrossPVal: INT;
	TON_6: TON;
	step2: INT;
	bAUnitBConeCrossing_1: BOOL;
	bAUnitBConeCrossedOff: BOOL;
	R_TRIG_3: R_TRIG;
	TON_8: TON;
	R_TRIG_11: R_TRIG;

	F_TRIG_4: F_TRIG;
	tRowStopperMidDly2: TON;
	tUnitBCountDelay1: TON;
	ConeInCompleteB: BOOL;
	TEnableCounterB: BOOL;
	CompleteTestbitB: BOOL;
	bCounterDisableUnitB: BOOL;
	TestTimer: TON;
	bStartUnitBCompCount: BOOL;
	step3: INT;
	F_TRIG_5: F_TRIG;
	TON_9: TON;
	TON_10: TON;
	TON_11: TON;
	TON_12: TON;
	bAUnitBConeCrossedTemp: BOOL;
END_VAR
(*=============CHecking the No of sensors sensed on conveyor ==================*)

IF bCheckSensor THEN
SenSelect_2(
		bVarIn1:=bIUnitBConeDetection1 ,
		bVarIn2:= bIUnitBConeDetection2,
		bVarIn3:= bIUnitBConeDetection3,
		bVarIn4:= bIUnitBConeDetection4,
		ByteResult=>iSensorOnVal );


END_IF

IF iSensorOnVal=15 THEN iAConeCrossCount:=4;
		ELSIF  iSensorOnVal=14 THEN iAConeCrossCount:=3;
		ELSIF  iSensorOnVal=13 THEN iAConeCrossCount:=3;
		ELSIF  iSensorOnVal=12 THEN iAConeCrossCount:=2;
		ELSIF  iSensorOnVal=11 THEN iAConeCrossCount:=3;
		ELSIF  iSensorOnVal=10 THEN iAConeCrossCount:=2;
		ELSIF  iSensorOnVal=9 THEN iAConeCrossCount:=2;
		ELSIF  iSensorOnVal=8 THEN iAConeCrossCount:=1;
		ELSIF  iSensorOnVal=7 THEN iAConeCrossCount:=3;
		ELSIF  iSensorOnVal=6 THEN iAConeCrossCount:=2;
		ELSIF  iSensorOnVal=5 THEN iAConeCrossCount:=2;
		ELSIF  iSensorOnVal=4 THEN iAConeCrossCount:=1;
		ELSIF  iSensorOnVal=3 THEN iAConeCrossCount:=2;
		ELSIF  iSensorOnVal=2 THEN iAConeCrossCount:=1;
		ELSIF  iSensorOnVal=1 THEN iAConeCrossCount:=1;
		END_IF





bQAUnitBRowStopperMotorFwd:=( bQAUnitB_RowStopperMotorFwd1  );

bQAUnitBRowStopperMotorRev:= ( bQAUnitB_RowStopperMotorRev1 OR bRetUnitBRst  );

CASE step OF

	0:	CycleComplete1:=FALSE;
		IF bAutoModeOn  AND bAUnitBWeighOk  AND bRetUnitBStart  AND NOT bAInializeStarted AND NOT bIntialAckBit AND bInterlockInitial_2  THEN
		UnitBConeCrossCount.RESET:=TRUE;

		CTU_2.RESET:=TRUE;
		step:=step+1;
		END_IF

	1:
		step:=step+1;

	2:	IF bAutoModeOn(* AND bIUnitB_LiftPistonHome *)THEN
		CTU_2.RESET:=FALSE;
		UnitBConeCrossCount.RESET:=FALSE;
		UnitBCompleteCheckCount.RESET:=FALSE;
		step:=step+1;
		END_IF


	3:	UnitBConeCompChkCount.RESET:=FALSE;
		TestTimer(IN:=FALSE);
		step:=step+1;


	4:	IF bAutoModeOn   AND NOT  bUnitARowStopperStarted  AND NOT ConeInCompleteA AND NOT  ConeInCompleteB  AND NOT bAPauseSeq
		(*AND NOT bIUnitBConedetection1 AND NOT bIUnitBConedetection2 AND NOT bIUnitBConedetection3 *) AND bInterlockInitial_2 THEN
		timer1(IN:=FALSE);
		timer2(IN:=FALSE);
		bQAUnitB_RowStopperMotorFwd1:=TRUE;
		bAUnitBWeighOk:=FALSE;
		sRetreivalBStatus:= 'Running';
		bUnitBRowStopperStarted:=TRUE;
	(*	UnitBConeCrossCount.RESET:=TRUE; *)

		step:=step+1;
		END_IF

	5:	RowStopperMotorStopDly(In:=FALSE); step:=step+1;


	6:	IF bIUnitBConedetection1 OR  bIUnitBConedetection2  OR  bIUnitBConedetection3  OR bIUnitBConedetection4  AND NOT bAPauseSeq THEN

		step:=step+1;
		ELSIF NOT bIUnitBConedetection1 AND NOT  bIUnitBConedetection2 AND NOT  bIUnitBConedetection3 AND NOT bIUnitBConedetection4  AND bIUnitB_RowStopperEnd THEN

		step:=15;

		END_IF

	7:	CompleteTestbitB:=FALSE;
		UnitBConeCompChkCount.RESET:=TRUE;
		RowStopperMotorStopDly( IN:=TRUE , PT:=T#0.4S , Q=> , ET=> );
		IF RowStopperMotorStopDly.Q   THEN UnitBConeCrossCount.RESET:=FALSE;  UnitBConeCompChkCount.RESET:=FALSE ; step:=step+1; END_IF


	8:	bStartUnitBCompCount:=TRUE;
		bQAUnitB_RowStopperMotorFwd1:=FALSE;
		tRowStopperRevDly1(IN:=FALSE);
		GetDLy(IN:=FALSE);
		step:=step+1;

	9:	IF NOT   bAPauseSeq THEN bCheckSensor:=TRUE; step:=step+1;END_IF

	10:	GetDLy(IN:=TRUE , PT:=t#0.4s , Q=> , ET=> );
		 IF GetDLy.Q THEN bCheckSensor:=FALSE;  tConeChkDly(IN:=FALSE);  step:=step+1;
		END_IF



	11:	IF UnitBConeCrossCount.CV>=iAConeCrossCount  THEN
		RowStopperMotorStopDly(In:=FALSE);
		 tConeChkDly(IN:=FALSE);
		GetDLy(IN:=FALSE);
		step:=step+1;
		ELSIF UnitBConeCrossCount.CV <> iAConeCrossCount  THEN
		tConeChkDly(IN:=TRUE , PT:=t#5s , Q=> , ET=> );
	(*	IF tConeChkDly.Q THEN bConeMiss:=TRUE; ELSE bConeMiss:=FALSE ;  END_IF *)
		END_IF


	12:	IF NOT bAPauseSeq THEN tRowStopperRevDly1(IN:=FALSE); step:=step+1; END_IF

	13:	IF bAutoModeOn   THEN
		UnitBConeCrossCount.RESET:=TRUE;
		step:=step+1;
		END_IF


	14:	 UnitBConeCrossCount.RESET:=FALSE; step:=step+1;

	15:	IF bAutoModeOn AND bIUnitB_RowStopperEnd THEN
		bQAUnitB_RowStopperMotorFwd1:=FALSE;
		 step:=step+1;
		ELSIF  bAutoModeOn AND NOT  bIUnitB_RowStopperEnd  THEN
		 step:=4;
		END_IF

	16:	tRowStopperRevDly1(IN:=TRUE , PT:=t#1.5s , Q=> , ET=> );
		IF tRowStopperRevDly1.Q THEN step:=step+1; END_IF

	17:	step:=step+1;

